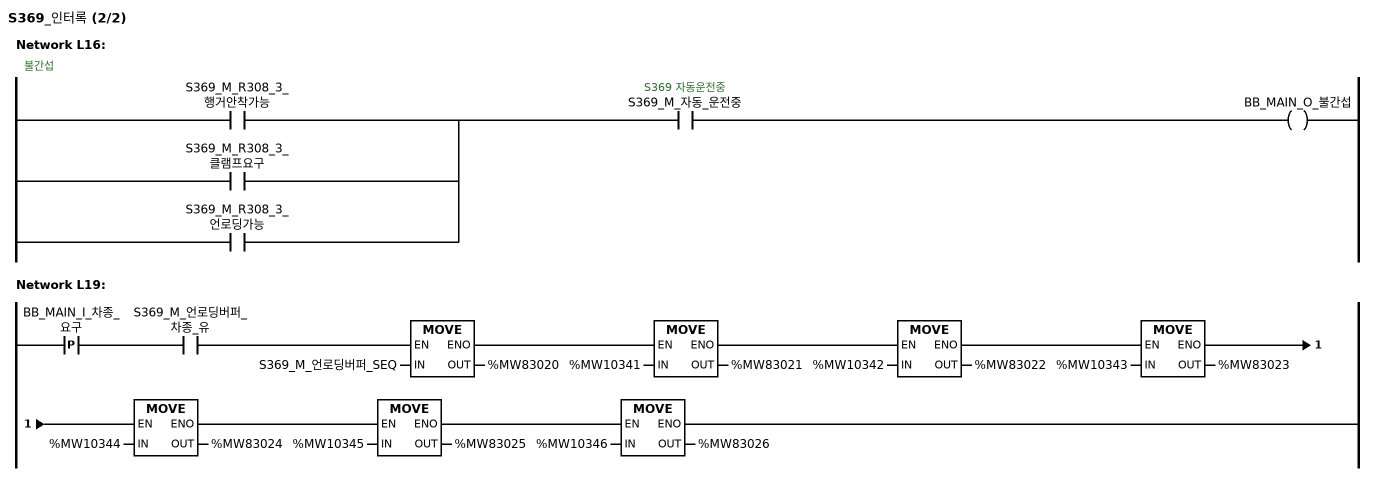
(* [picture p312: S369_인터록 rungs L16-L19] *)
(* 불간섭 *)
(* Rung L16 *)
BB_MAIN_O_불간섭 := (S369_M_R308_3_행거안착가능 OR S369_M_R308_3_클램프요구 OR S369_M_R308_3_언로딩가능) AND S369_M_자동_운전중;
(* Rung L19 *)
_e1(CLK := BB_MAIN_I_차종_요구);
IF _e1.Q AND S369_M_언로딩버퍼_차종_유 THEN
    %MW83020 := S369_M_언로딩버퍼_SEQ;
    %MW83021 := %MW10341;
    %MW83022 := %MW10342;
    %MW83023 := %MW10343;
    %MW83024 := %MW10344;
    %MW83025 := %MW10345;
    %MW83026 := %MW10346;
END_IF;
END_PROGRAM

PROGRAM S369_이상 (* task: 스캔 프로그램 *)
VAR
    INST10 : TON;
    INST11 : TON;
    INST12 : TON;
    INST13 : TON;
    INST14 : TON;
    INST15 : TON;
    INST16 : TON;
    INST17 : TON;
    INST18 : TON;
    INST19 : TON;
    INST20 : TON;
    INST21 : TON;
    INST22 : TON;
    INST23 : TON;
    INST24 : TON;
    INST25 : TON;
    INST26 : TON;
    INST27 : TON;
    INST28 : TON;
    INST29 : TON;
    INST30 : TON;
    INST31 : TON;
    INST32 : TON;
    INST33 : TON;
    INST34 : TON;
    INST35 : TON;
    INST36 : TON;
    INST37 : TON;
    INST38 : TON;
    INST8 : TON;
    INST9 : TON;
END_VAR
VAR_EXTERNAL RETAIN
    S368_M_공정_불간섭 : BOOL; (* AT %MW4004.1 *) (* S368_M_공정_불간섭 *)
    S368_M_공정_제품감지_무 : BOOL; (* AT %MW4001.6 *) (* S368_M_공정_제품감지_무 *)
    S368_M_공정_차종_유 : BOOL; (* AT %MW4002.0 *) (* S368_M_공정_차종_유 *)
    S368_M_자동_운전중 : BOOL; (* AT %MW4000.4 *) (* S368 자동운전중 *)
    S369_LOAD_M_NODE_6_41_통신_이상 : BOOL; (* AT %MW5024.0 *)
    S369_M_LD_CP_OFF : BOOL; (* AT %MW5017.0 *) (* S369_M_LD_CP_OFF *)
    S369_M_LD_EJECT_상승_LS_이상 : BOOL; (* AT %MW5100.5 *) (* S369_M_LD_EJECT_상승_LS_이상 *)
    S369_M_LD_EJECT_제품감지_이상 : BOOL; (* AT %MW5014.0 *) (* S369_M_LD_제품감지_이상 *)
    S369_M_LD_EJECT_하강_LS_이상 : BOOL; (* AT %MW5100.6 *) (* S369_M_LD_EJECT_하강_LS_이상 *)
    S369_M_LD_LH_LAT_전진_LS_이상 : BOOL; (* AT %MW5101.5 *) (* S369_M_LD_LH_LAT_전진_LS_이상 *)
    S369_M_LD_LH_LAT_후진_LS_이상 : BOOL; (* AT %MW5101.6 *) (* S369_M_LD_LH_LAT_후진_LS_이상 *)
    S369_M_LD_RH_LAT_전진_LS_이상 : BOOL; (* AT %MW5102.5 *) (* S369_M_LD_RH_LAT_전진_LS_이상 *)
    S369_M_LD_RH_LAT_후진_LS_이상 : BOOL; (* AT %MW5102.6 *) (* S369_M_LD_RH_LAT_후진_LS_이상 *)
    S369_M_LD_공기압_이상 : BOOL; (* AT %MW5013.0 *) (* S369_M_LD_공기압_이상 *)
    S369_M_LD_차종_이상 : BOOL; (* AT %MW5015.0 *) (* S369_M_LD_차종_이상 *)
    S369_M_R308_3_언로딩완료 : BOOL; (* AT %MW5001.5 *)
    S369_M_R369_2_로딩가능 : BOOL; (* AT %MW5004.8 *)
    S369_M_R369_2_로딩완료 : BOOL; (* AT %MW5001.2 *)
    S369_M_SERVO_DRIVE_통신이상 : BOOL; (* AT %MW5024.8 *)
    S369_M_SRV_NFB_OFF : BOOL; (* AT %MW5021.0 *) (* S369_M_SRV_NFB_OFF *)
    S369_M_UD_CP_OFF : BOOL; (* AT %MW5017.1 *) (* S369_M_UD_CP_OFF *)
    S369_M_UD_DOCK_CLP_전진_LS_이상 : BOOL; (* AT %MW5111.5 *) (* S369_M_UD_DOCK_CLP_전진_LS_이상 *)
    S369_M_UD_DOCK_CLP_후진_LS_이상 : BOOL; (* AT %MW5111.6 *) (* S369_M_UD_DOCK_CLP_후진_LS_이상 *)
    S369_M_UD_EJECT_상승_LS_이상 : BOOL; (* AT %MW5108.5 *) (* S369_M_UD_EJECT_상승_LS_이상 *)
    S369_M_UD_EJECT_상승단 : BOOL; (* AT %MW5108.3 *) (* S369_M_UD_EJECT_상승단 *)
    S369_M_UD_EJECT_제품감지_이상 : BOOL; (* AT %MW5014.1 *) (* S369_M_UD_제품감지_이상 *)
    S369_M_UD_EJECT_하강_LS_이상 : BOOL; (* AT %MW5108.6 *) (* S369_M_UD_EJECT_하강_LS_이상 *)
    S369_M_UD_LH_LAT_전진_LS_이상 : BOOL; (* AT %MW5109.5 *) (* S369_M_UD_LH_LAT_전진_LS_이상 *)
    S369_M_UD_LH_LAT_전진단 : BOOL; (* AT %MW5109.3 *) (* S369_M_UD_LH_LAT_전진단 *)
    S369_M_UD_LH_LAT_후진_LS_이상 : BOOL; (* AT %MW5109.6 *) (* S369_M_UD_LH_LAT_후진_LS_이상 *)
    S369_M_UD_RH_LAT_전진_LS_이상 : BOOL; (* AT %MW5110.5 *) (* S369_M_UD_RH_LAT_전진_LS_이상 *)
    S369_M_UD_RH_LAT_전진단 : BOOL; (* AT %MW5110.3 *) (* S369_M_UD_RH_LAT_전진단 *)
    S369_M_UD_RH_LAT_후진_LS_이상 : BOOL; (* AT %MW5110.6 *) (* S369_M_UD_RH_LAT_후진_LS_이상 *)
    S369_M_UD_공기압_이상 : BOOL; (* AT %MW5013.1 *) (* S369_M_UD_공기압_이상 *)
    S369_M_UD_차종_이상 : BOOL; (* AT %MW5015.1 *) (* S369_M_UD_차종_이상 *)
    S369_M_로딩_공정_불간섭 : BOOL; (* AT %MW5004.2 *) (* S369_M_공정_불간섭 *)
    S369_M_로딩_이젝터_제품감지_무 : BOOL; (* AT %MW5001.9 *)
    S369_M_로딩_이젝터_제품감지_유 : BOOL; (* AT %MW5001.8 *)
    S369_M_로딩버퍼_차종_유 : BOOL; (* AT %MW5002.0 *)
    S369_M_언로딩_공정_불간섭 : BOOL; (* AT %MW5004.3 *)
    S369_M_언로딩_이젝터_제품감지_무 : BOOL; (* AT %MW5001.11 *)
    S369_M_언로딩_이젝터_제품감지_유 : BOOL; (* AT %MW5001.10 *)
    S369_M_언로딩버퍼_차종_유 : BOOL; (* AT %MW5002.2 *)
    S369_M_이송버퍼1_제품감지_이상 : BOOL; (* AT %MW5014.5 *) (* S369_M_BELT4_제품감지_이상 *)
    S369_M_이송버퍼2_제품감지_이상 : BOOL; (* AT %MW5014.4 *) (* S369_M_BELT3_제품감지_이상 *)
    S369_M_이송버퍼3_제품감지_이상 : BOOL; (* AT %MW5014.3 *) (* S369_M_BELT2_제품감지_이상 *)
    S369_M_이송버퍼4_제품감지_이상 : BOOL; (* AT %MW5014.2 *) (* S369_M_BELT1_제품감지_이상 *)
    S369_M_자동_운전중 : BOOL; (* AT %MW5000.4 *) (* S369 자동운전중 *)
    S369_M_총괄_CP_이상 : BOOL; (* AT %MW5009.7 *) (* S369 CP OFF 이상 *)
    S369_M_총괄_CT_이상 : BOOL; (* AT %MW5010.4 *) (* S369   TACK TIME 이상 *)
    S369_M_총괄_EOCR_이상 : BOOL; (* AT %MW5009.8 *) (* S369_M_총괄_EOCR_이상 *)
    S369_M_총괄_INV_이상 : BOOL; (* AT %MW5009.9 *) (* S369_M_총괄_INV_이상 *)
    S369_M_총괄_LS_이상 : BOOL; (* AT %MW5009.15 *) (* S369 LS 이상 *)
    S369_M_총괄_MATCH_이상 : BOOL; (* AT %MW5010.0 *) (* S369 매트SW 이상 *)
    S369_M_총괄_MC_이상 : BOOL; (* AT %MW5009.13 *) (* S369_M_총괄_MC_이상 *)
    S369_M_총괄_NFB_이상 : BOOL; (* AT %MW5009.11 *) (* S369 NFB 이상 *)
    S369_M_총괄_ROBOT_이상 : BOOL; (* AT %MW5010.1 *) (* S369 ROBOT 이상 *)
    S369_M_총괄_SAFETY_이상 : BOOL; (* AT %MW5009.2 *) (* S369_M_총괄_SAFETY_이상 *)
    S369_M_총괄_SRV_이상 : BOOL; (* AT %MW5009.10 *) (* S369 SERVO 이상 *)
    S369_M_총괄_공기압_이상 : BOOL; (* AT %MW5009.3 *) (* S369 공기압 이상 *)
    S369_M_총괄_사양_이상 : BOOL; (* AT %MW5009.6 *) (* S369 사양 이상 *)
    S369_M_총괄_오버런_이상 : BOOL; (* AT %MW5009.12 *) (* S369 OVER RUN 이상 *)
    S369_M_총괄_용접타점수_이상 : BOOL; (* AT %MW5010.2 *) (* S369 용접타점수 이상 *)
    S369_M_총괄_이상 : BOOL; (* AT %MW5009.0 *) (* S369_M_총괄_이상 *)
    S369_M_총괄_제품감지_이상 : BOOL; (* AT %MW5009.4 *) (* S369 제품감지 이상 *)
    S369_M_총괄_차종_이상 : BOOL; (* AT %MW5009.5 *) (* S369 차종 이상 *)
    S369_M_총괄_통신_이상 : BOOL; (* AT %MW5009.14 *) (* S369 통신이상 *)
    S369_M_컨베어_MC_이상 : BOOL; (* AT %MW5023.0 *)
    S369_UNLD_M_NODE_6_42_통신_이상 : BOOL; (* AT %MW5024.1 *)
    전체_M_이상_리셋 : BOOL; (* AT %MW308.2 *) (* ALL공정 PB 이상리셋 *)
END_VAR
VAR_EXTERNAL
    S369LD_6_41_PLC_BOX_CP_TRIP : BOOL; (* AT %MW86412.15 *) (* S369LD_6_41_PLC_BOX_CP_TRIP *)
    S369LD_공기압_AIR_CHECK : BOOL; (* AT %MW86412.14 *) (* S369LD_공기압_AIR_CHECK *)
    S369UD_6_42_PLC_BOX_CP_TRIP : BOOL; (* AT %MW86422.15 *) (* S369UD_6_42_PLC_BOX_CP_TRIP *)
    S369UD_공기압_AIR_CHECK : BOOL; (* AT %MW86422.14 *) (* S369UD_공기압_AIR_CHECK *)
    S369_CONVEY_I_서보드라이브_이상 : BOOL; (* AT %MW50000.8 *)
    S369_SERVO_MC_ON : BOOL; (* AT %MW85022.0 *) (* SERVO_BRAKE_ON *)
    S369_SERVO_NFB_ON : BOOL; (* AT %MW85023.0 *)
    SERVO_SAFETY_CR_ON : BOOL; (* AT %MW95024.0 *) (* SERVO_BRAKE_CR_ON *)
    _0005_EB63_S00_SVC_ER : BOOL; (* AT %MW185036.7 *) (* 통신 서비스 에러 *)
    _0006_EB41_CFG_ER : BOOL; (* AT %MW186064.0 *) (* EB 구성 에러 *)
    _0006_EB41_DEER : BOOL; (* AT %MW186064.1 *) (* EB 운전 중 탈락 *)
    _0006_EB41_IO_DEER : BOOL; (* AT %MW186065.2 *) (* EB IO 탈락 에러 *)
    _0006_EB41_IO_TYER : BOOL; (* AT %MW186065.1 *) (* EB IO 타입 에러 *)
    _0006_EB42_CFG_ER : BOOL; (* AT %MW186070.0 *) (* EB 구성 에러 *)
    _0006_EB42_DEER : BOOL; (* AT %MW186070.1 *) (* EB 운전 중 탈락 *)
    _0006_EB42_IO_DEER : BOOL; (* AT %MW186071.2 *) (* EB IO 탈락 에러 *)
    _0006_EB42_IO_TYER : BOOL; (* AT %MW186071.1 *) (* EB IO 타입 에러 *)
    _0007_EB10_CFG_ER : BOOL; (* AT %MW187040.0 *) (* EB 구성 에러 *)
    _0007_EB10_DEER : BOOL; (* AT %MW187040.1 *) (* EB 운전 중 탈락 *)
    _0007_EB10_IO_DEER : BOOL; (* AT %MW187041.2 *) (* EB IO 탈락 에러 *)
    _0007_EB10_IO_TYER : BOOL; (* AT %MW187041.1 *) (* EB IO 타입 에러 *)
END_VAR

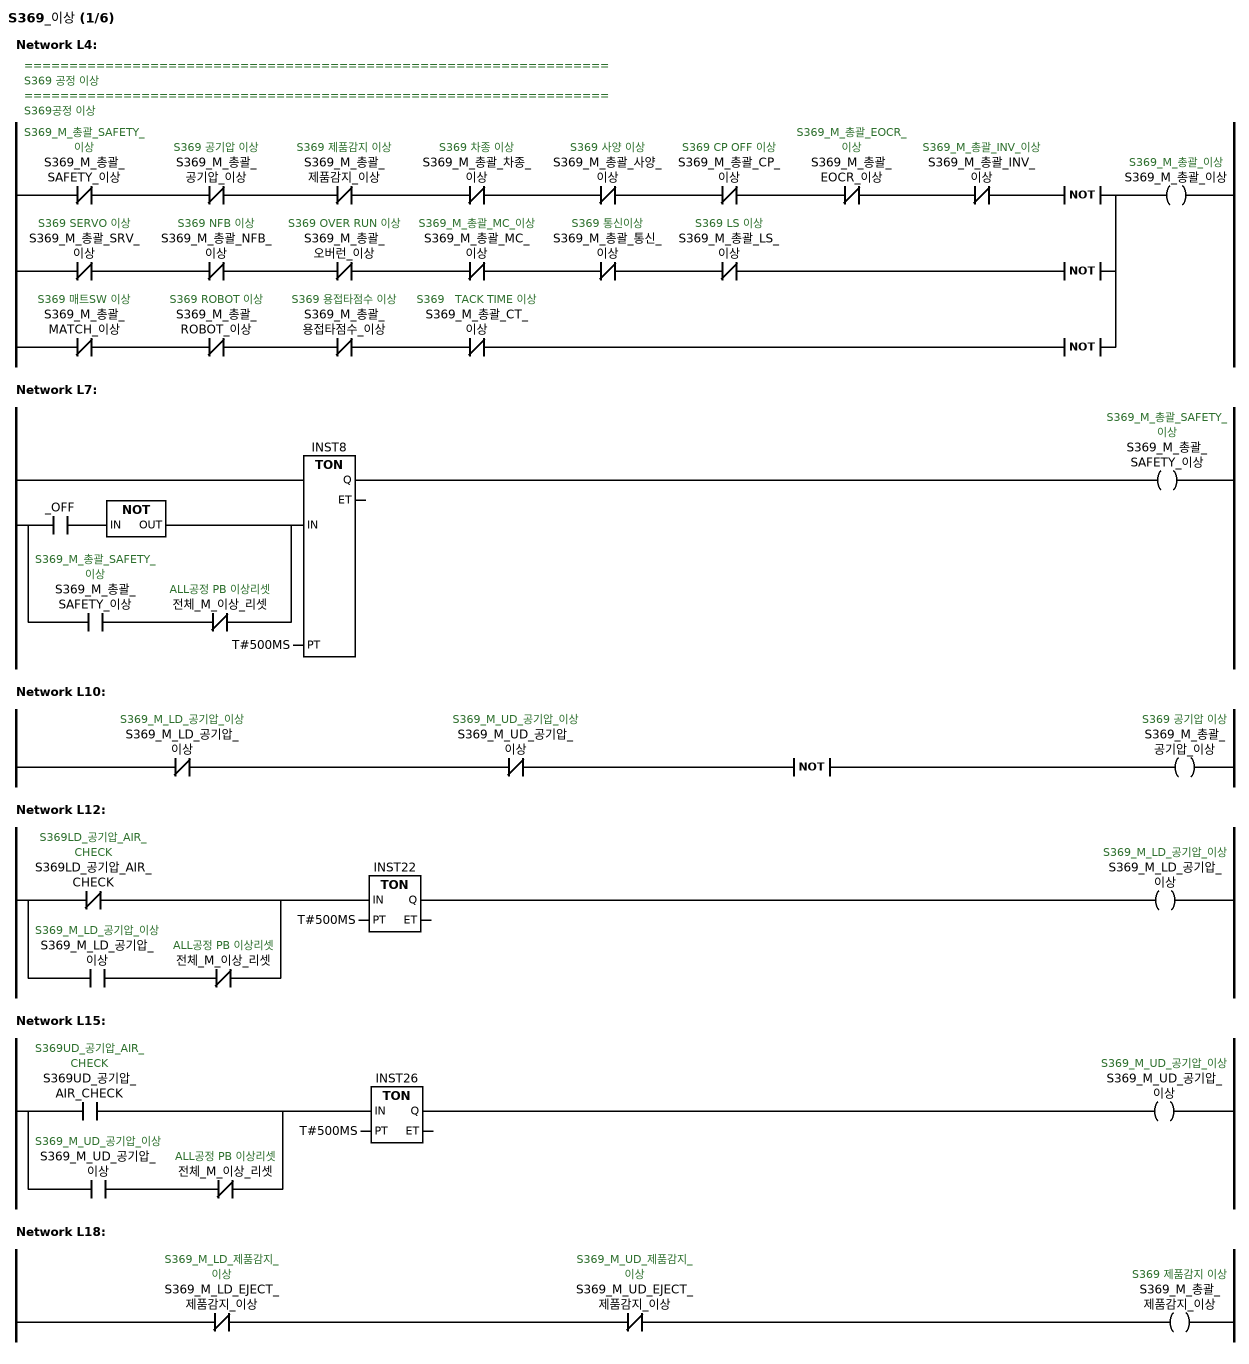
(* ================================================================= *)
(* S369 공정 이상 *)
(* ================================================================= *)
(* S369공정 이상 *)
(* Rung L4 *)
S369_M_총괄_이상 := NOT (NOT S369_M_총괄_SAFETY_이상 AND NOT S369_M_총괄_공기압_이상 AND NOT S369_M_총괄_제품감지_이상 AND NOT S369_M_총괄_차종_이상 AND NOT S369_M_총괄_사양_이상 AND NOT S369_M_총괄_CP_이상 AND NOT S369_M_총괄_EOCR_이상 AND NOT S369_M_총괄_INV_이상) OR NOT (NOT S369_M_총괄_SRV_이상 AND NOT S369_M_총괄_NFB_이상 AND NOT S369_M_총괄_오버런_이상 AND NOT S369_M_총괄_MC_이상 AND NOT S369_M_총괄_통신_이상 AND NOT S369_M_총괄_LS_이상) OR NOT (NOT S369_M_총괄_MATCH_이상 AND NOT S369_M_총괄_ROBOT_이상 AND NOT S369_M_총괄_용접타점수_이상 AND NOT S369_M_총괄_CT_이상);
(* Rung L7 *)
INST8(IN := (NOT _OFF) OR (S369_M_총괄_SAFETY_이상 AND NOT 전체_M_이상_리셋), PT := T#500MS);
S369_M_총괄_SAFETY_이상 := INST8.Q;
(* Rung L10 *)
S369_M_총괄_공기압_이상 := NOT (NOT S369_M_LD_공기압_이상 AND NOT S369_M_UD_공기압_이상);
(* Rung L12 *)
INST22(IN := NOT S369LD_공기압_AIR_CHECK OR (S369_M_LD_공기압_이상 AND NOT 전체_M_이상_리셋), PT := T#500MS);
S369_M_LD_공기압_이상 := INST22.Q;
(* Rung L15 *)
INST26(IN := S369UD_공기압_AIR_CHECK OR (S369_M_UD_공기압_이상 AND NOT 전체_M_이상_리셋), PT := T#500MS);
S369_M_UD_공기압_이상 := INST26.Q;
(* Rung L18 *)
S369_M_총괄_제품감지_이상 := NOT S369_M_LD_EJECT_제품감지_이상 AND NOT S369_M_UD_EJECT_제품감지_이상;

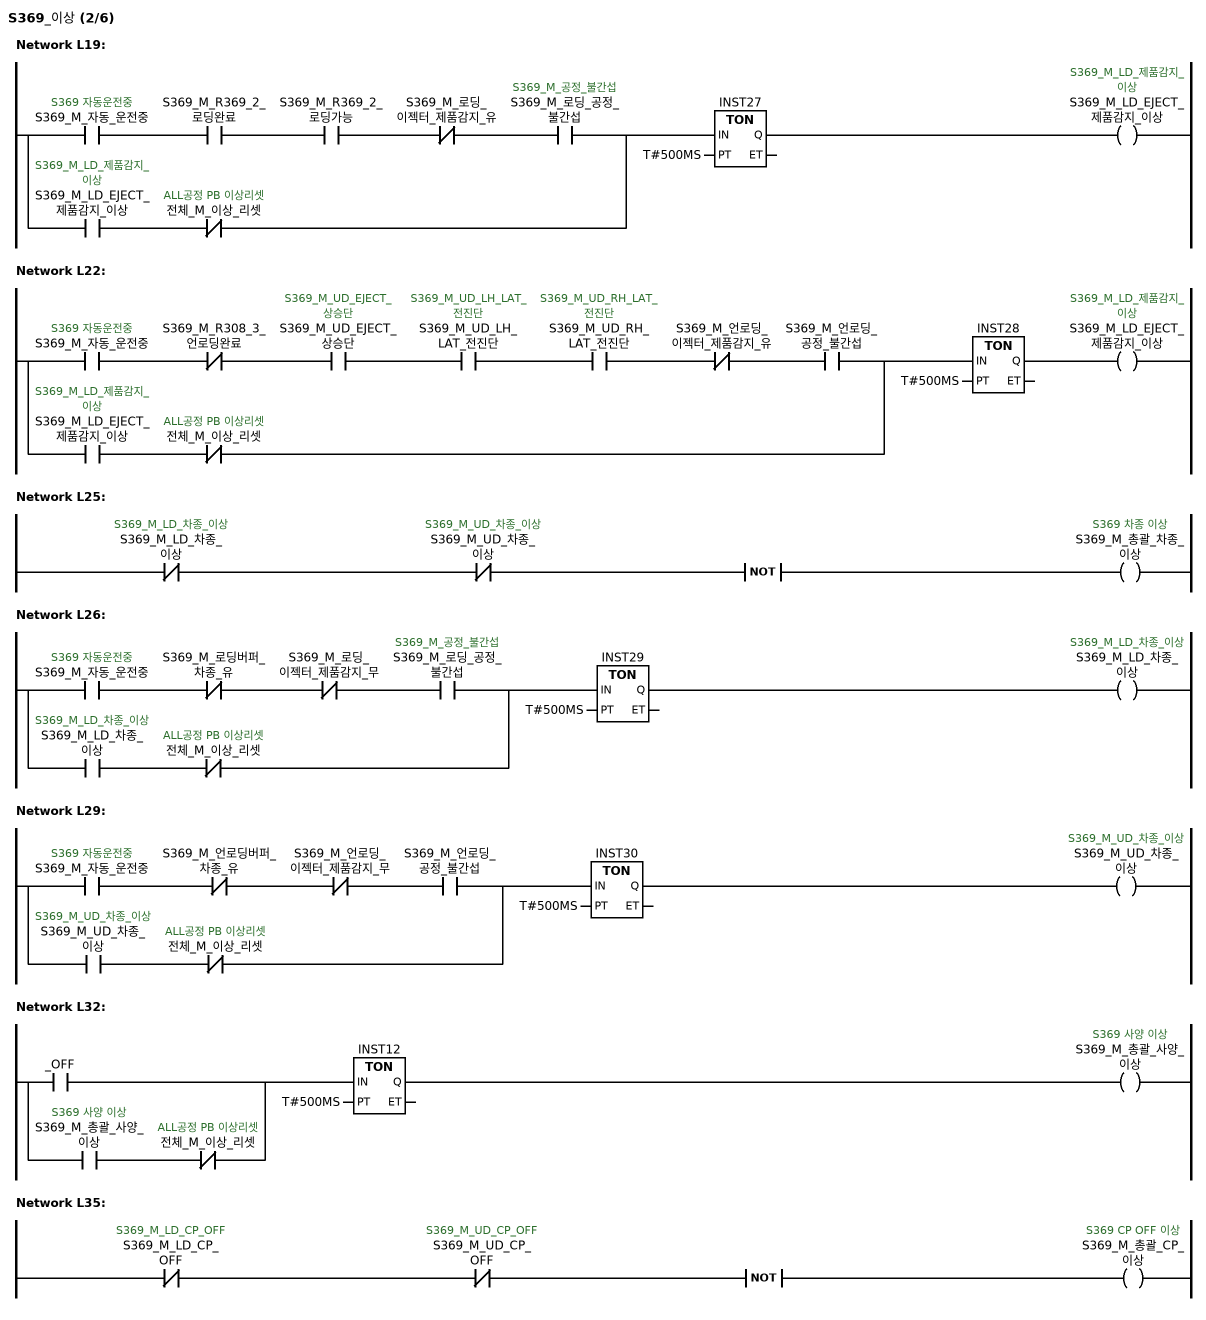
(* Rung L19 *)
INST27(IN := (S369_M_자동_운전중 AND S369_M_R369_2_로딩완료 AND S369_M_R369_2_로딩가능 AND NOT S369_M_로딩_이젝터_제품감지_유 AND S369_M_로딩_공정_불간섭) OR (S369_M_LD_EJECT_제품감지_이상 AND NOT 전체_M_이상_리셋), PT := T#500MS);
S369_M_LD_EJECT_제품감지_이상 := INST27.Q;
(* Rung L22 *)
INST28(IN := (S369_M_자동_운전중 AND NOT S369_M_R308_3_언로딩완료 AND S369_M_UD_EJECT_상승단 AND S369_M_UD_LH_LAT_전진단 AND S369_M_UD_RH_LAT_전진단 AND NOT S369_M_언로딩_이젝터_제품감지_유 AND S369_M_언로딩_공정_불간섭) OR (S369_M_LD_EJECT_제품감지_이상 AND NOT 전체_M_이상_리셋), PT := T#500MS);
S369_M_LD_EJECT_제품감지_이상 := INST28.Q;
(* Rung L25 *)
S369_M_총괄_차종_이상 := NOT (NOT S369_M_LD_차종_이상 AND NOT S369_M_UD_차종_이상);
(* Rung L26 *)
INST29(IN := (S369_M_자동_운전중 AND NOT S369_M_로딩버퍼_차종_유 AND NOT S369_M_로딩_이젝터_제품감지_무 AND S369_M_로딩_공정_불간섭) OR (S369_M_LD_차종_이상 AND NOT 전체_M_이상_리셋), PT := T#500MS);
S369_M_LD_차종_이상 := INST29.Q;
(* Rung L29 *)
INST30(IN := (S369_M_자동_운전중 AND NOT S369_M_언로딩버퍼_차종_유 AND NOT S369_M_언로딩_이젝터_제품감지_무 AND S369_M_언로딩_공정_불간섭) OR (S369_M_UD_차종_이상 AND NOT 전체_M_이상_리셋), PT := T#500MS);
S369_M_UD_차종_이상 := INST30.Q;
(* Rung L32 *)
INST12(IN := _OFF OR (S369_M_총괄_사양_이상 AND NOT 전체_M_이상_리셋), PT := T#500MS);
S369_M_총괄_사양_이상 := INST12.Q;
(* Rung L35 *)
S369_M_총괄_CP_이상 := NOT (NOT S369_M_LD_CP_OFF AND NOT S369_M_UD_CP_OFF);

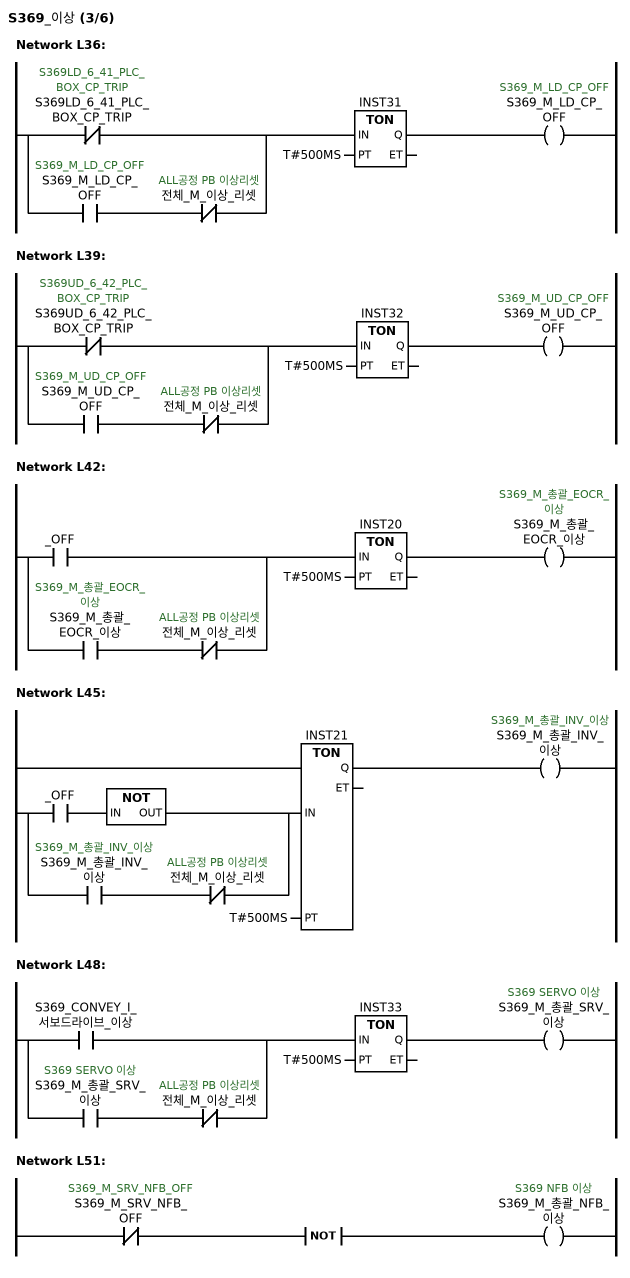
(* Rung L36 *)
INST31(IN := NOT S369LD_6_41_PLC_BOX_CP_TRIP OR (S369_M_LD_CP_OFF AND NOT 전체_M_이상_리셋), PT := T#500MS);
S369_M_LD_CP_OFF := INST31.Q;
(* Rung L39 *)
INST32(IN := NOT S369UD_6_42_PLC_BOX_CP_TRIP OR (S369_M_UD_CP_OFF AND NOT 전체_M_이상_리셋), PT := T#500MS);
S369_M_UD_CP_OFF := INST32.Q;
(* Rung L42 *)
INST20(IN := _OFF OR (S369_M_총괄_EOCR_이상 AND NOT 전체_M_이상_리셋), PT := T#500MS);
S369_M_총괄_EOCR_이상 := INST20.Q;
(* Rung L45 *)
INST21(IN := (NOT _OFF) OR (S369_M_총괄_INV_이상 AND NOT 전체_M_이상_리셋), PT := T#500MS);
S369_M_총괄_INV_이상 := INST21.Q;
(* Rung L48 *)
INST33(IN := S369_CONVEY_I_서보드라이브_이상 OR (S369_M_총괄_SRV_이상 AND NOT 전체_M_이상_리셋), PT := T#500MS);
S369_M_총괄_SRV_이상 := INST33.Q;
(* Rung L51 *)
S369_M_총괄_NFB_이상 := S369_M_SRV_NFB_OFF;

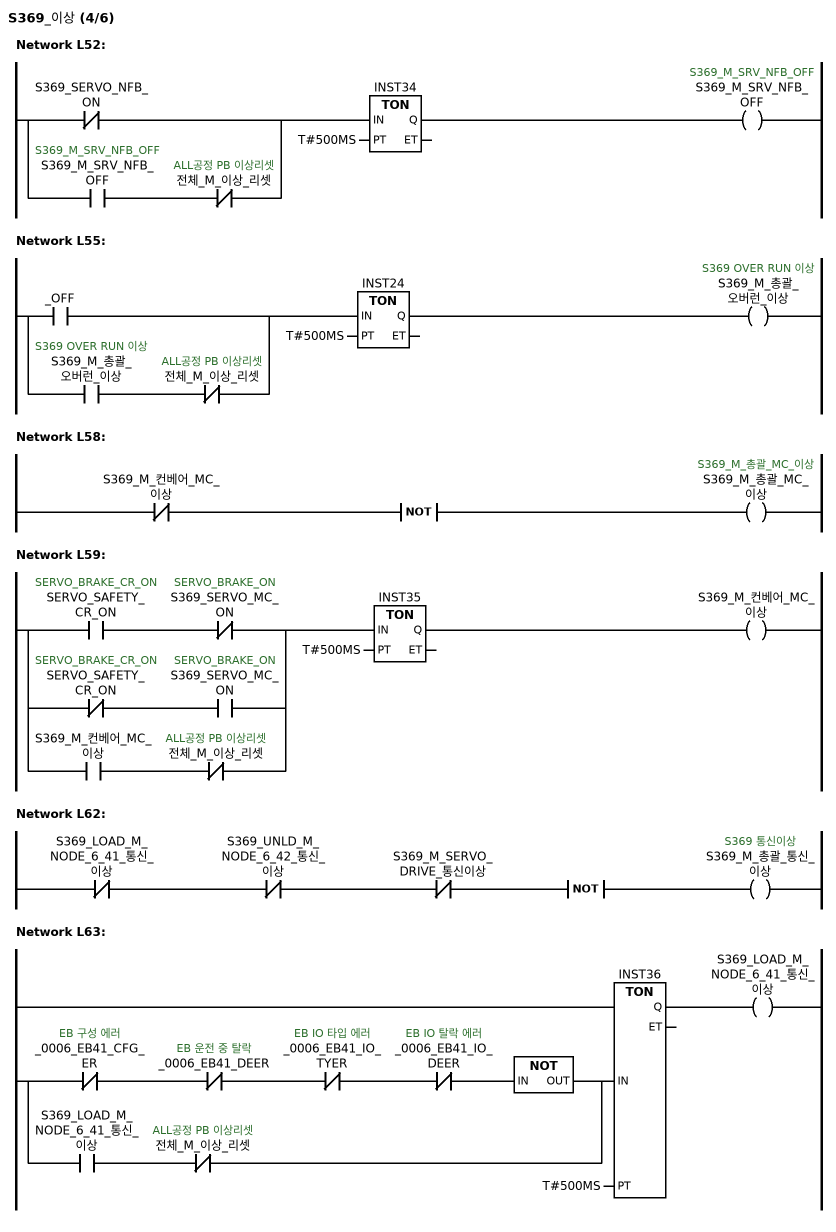
(* Rung L52 *)
INST34(IN := NOT S369_SERVO_NFB_ON OR (S369_M_SRV_NFB_OFF AND NOT 전체_M_이상_리셋), PT := T#500MS);
S369_M_SRV_NFB_OFF := INST34.Q;
(* Rung L55 *)
INST24(IN := _OFF OR (S369_M_총괄_오버런_이상 AND NOT 전체_M_이상_리셋), PT := T#500MS);
S369_M_총괄_오버런_이상 := INST24.Q;
(* Rung L58 *)
S369_M_총괄_MC_이상 := S369_M_컨베어_MC_이상;
(* Rung L59 *)
INST35(IN := (SERVO_SAFETY_CR_ON AND NOT S369_SERVO_MC_ON) OR (NOT SERVO_SAFETY_CR_ON AND S369_SERVO_MC_ON) OR (S369_M_컨베어_MC_이상 AND NOT 전체_M_이상_리셋), PT := T#500MS);
S369_M_컨베어_MC_이상 := INST35.Q;
(* Rung L62 *)
S369_M_총괄_통신_이상 := NOT (NOT S369_LOAD_M_NODE_6_41_통신_이상 AND NOT S369_UNLD_M_NODE_6_42_통신_이상 AND NOT S369_M_SERVO_DRIVE_통신이상);
(* Rung L63 *)
INST36(IN := (NOT (NOT _0006_EB41_CFG_ER AND NOT _0006_EB41_DEER AND NOT _0006_EB41_IO_TYER AND NOT _0006_EB41_IO_DEER)) OR (S369_LOAD_M_NODE_6_41_통신_이상 AND NOT 전체_M_이상_리셋), PT := T#500MS);
S369_LOAD_M_NODE_6_41_통신_이상 := INST36.Q;

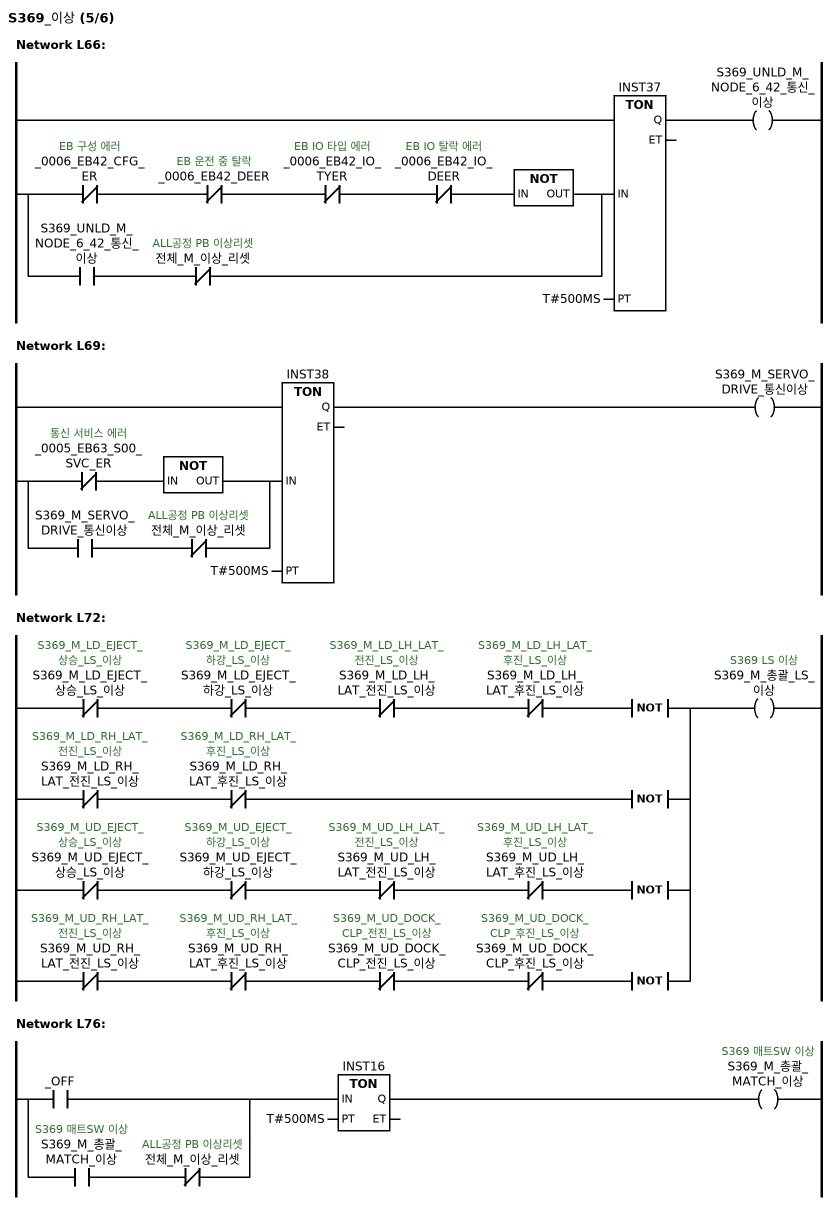
(* Rung L66 *)
INST37(IN := (NOT (NOT _0006_EB42_CFG_ER AND NOT _0006_EB42_DEER AND NOT _0006_EB42_IO_TYER AND NOT _0006_EB42_IO_DEER)) OR (S369_UNLD_M_NODE_6_42_통신_이상 AND NOT 전체_M_이상_리셋), PT := T#500MS);
S369_UNLD_M_NODE_6_42_통신_이상 := INST37.Q;
(* Rung L69 *)
INST38(IN := (NOT (NOT _0005_EB63_S00_SVC_ER)) OR (S369_M_SERVO_DRIVE_통신이상 AND NOT 전체_M_이상_리셋), PT := T#500MS);
S369_M_SERVO_DRIVE_통신이상 := INST38.Q;
(* Rung L72 *)
S369_M_총괄_LS_이상 := NOT (NOT S369_M_LD_EJECT_상승_LS_이상 AND NOT S369_M_LD_EJECT_하강_LS_이상 AND NOT S369_M_LD_LH_LAT_전진_LS_이상 AND NOT S369_M_LD_LH_LAT_후진_LS_이상) OR NOT (NOT S369_M_LD_RH_LAT_전진_LS_이상 AND NOT S369_M_LD_RH_LAT_후진_LS_이상) OR NOT (NOT S369_M_UD_EJECT_상승_LS_이상 AND NOT S369_M_UD_EJECT_하강_LS_이상 AND NOT S369_M_UD_LH_LAT_전진_LS_이상 AND NOT S369_M_UD_LH_LAT_후진_LS_이상) OR NOT (NOT S369_M_UD_RH_LAT_전진_LS_이상 AND NOT S369_M_UD_RH_LAT_후진_LS_이상 AND NOT S369_M_UD_DOCK_CLP_전진_LS_이상 AND NOT S369_M_UD_DOCK_CLP_후진_LS_이상);
(* Rung L76 *)
INST16(IN := _OFF OR (S369_M_총괄_MATCH_이상 AND NOT 전체_M_이상_리셋), PT := T#500MS);
S369_M_총괄_MATCH_이상 := INST16.Q;

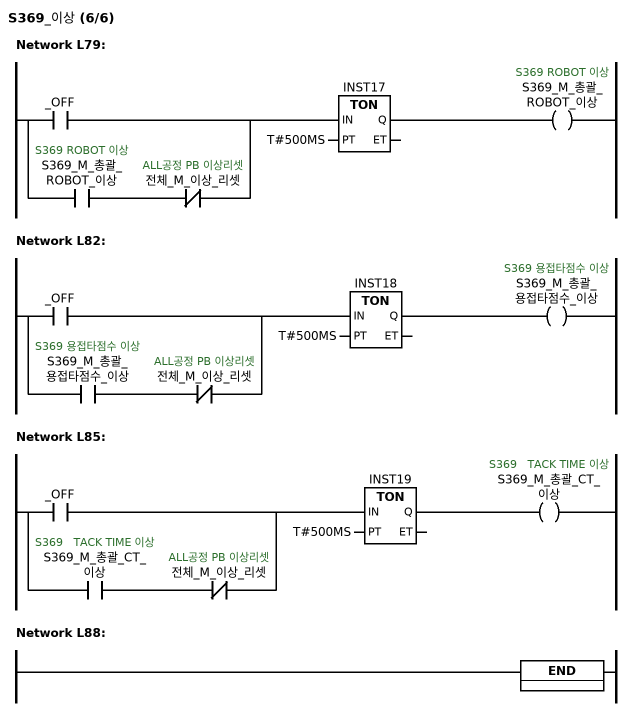
(* Rung L79 *)
INST17(IN := _OFF OR (S369_M_총괄_ROBOT_이상 AND NOT 전체_M_이상_리셋), PT := T#500MS);
S369_M_총괄_ROBOT_이상 := INST17.Q;
(* Rung L82 *)
INST18(IN := _OFF OR (S369_M_총괄_용접타점수_이상 AND NOT 전체_M_이상_리셋), PT := T#500MS);
S369_M_총괄_용접타점수_이상 := INST18.Q;
(* Rung L85 *)
INST19(IN := _OFF OR (S369_M_총괄_CT_이상 AND NOT 전체_M_이상_리셋), PT := T#500MS);
S369_M_총괄_CT_이상 := INST19.Q;
(* Rung L88 *)
END();
END_PROGRAM

PROGRAM HMI_차종수정 (* task: 스캔 프로그램 *)
VAR_EXTERNAL RETAIN
    CARTYPE : ARRAY[0..599] OF WORD; (* AT %MW10000 *) (* CARTYPE *)
    HMI_M_매칭_R361_1_S366 : BOOL; (* AT %MW70.0 *)
    HMI_M_매칭_S366_R361_1 : BOOL; (* AT %MW70.1 *)
    HMI_M_매칭선택 : WORD; (* AT %MW70 *)
    HMI_M_매칭차종_DATA_OK : BOOL; (* AT %MW9.9 *)
    HMI_M_매칭차종_복사_ON : BOOL; (* AT %MW9.6 *)
    HMI_M_매칭차종_복사_SET : BOOL; (* AT %MW9.8 *)
    HMI_M_차종매칭_SEQ : WORD; (* AT %MW50 *)
    HMI_M_차종매칭_차종1_AX : BOOL; (* AT %MW51.0 *)
    HMI_M_차종매칭_차종1_B : BOOL; (* AT %MW51.1 *)
    HMI_M_차종매칭_차종1_C : BOOL; (* AT %MW51.2 *)
    HMI_M_차종매칭_차종1_D : BOOL; (* AT %MW51.3 *)
    HMI_M_차종매칭_차종1_E : BOOL; (* AT %MW51.4 *)
    HMI_M_차종매칭_차종1_F : BOOL; (* AT %MW51.5 *)
    HMI_M_차종매칭_차종1_G : BOOL; (* AT %MW51.6 *)
    HMI_M_차종매칭_차종1_H : BOOL; (* AT %MW51.7 *)
    HMI_M_차종매칭_차종2_3DR : BOOL; (* AT %MW51.8 *)
    HMI_M_차종매칭_차종2_4DR : BOOL; (* AT %MW51.9 *)
    HMI_M_차종매칭_차종2_5DR : BOOL; (* AT %MW51.10 *)
    HMI_M_차종매칭_차종2_SP1 : BOOL; (* AT %MW51.12 *)
    HMI_M_차종매칭_차종2_SP2 : BOOL; (* AT %MW51.13 *)
    HMI_M_차종매칭_차종2_WGN : BOOL; (* AT %MW51.11 *)
    HMI_M_차종매칭_차종3_LHD : BOOL; (* AT %MW51.14 *)
    HMI_M_차종매칭_차종3_RHD : BOOL; (* AT %MW51.15 *)
    HMI_M_차종매칭_차종4_EEC : BOOL; (* AT %MW52.3 *)
    HMI_M_차종매칭_차종4_SP1 : BOOL; (* AT %MW52.8 *)
    HMI_M_차종매칭_차종4_SP2 : BOOL; (* AT %MW52.9 *)
    HMI_M_차종매칭_차종4_SP3 : BOOL; (* AT %MW52.11 *)
    HMI_M_차종매칭_차종4_SP4 : BOOL; (* AT %MW52.12 *)
    HMI_M_차종매칭_차종4_SP5 : BOOL; (* AT %MW52.13 *)
    HMI_M_차종매칭_차종4_SP6 : BOOL; (* AT %MW52.14 *)
    HMI_M_차종매칭_차종4_SP7 : BOOL; (* AT %MW52.15 *)
    HMI_M_차종매칭_차종4_내수 : BOOL; (* AT %MW52.0 *)
    HMI_M_차종매칭_차종4_러시아 : BOOL; (* AT %MW52.10 *)
    HMI_M_차종매칭_차종4_북미 : BOOL; (* AT %MW52.2 *)
    HMI_M_차종매칭_차종4_브라질 : BOOL; (* AT %MW52.7 *)
    HMI_M_차종매칭_차종4_수출 : BOOL; (* AT %MW52.1 *)
    HMI_M_차종매칭_차종4_중국 : BOOL; (* AT %MW52.6 *)
    HMI_M_차종매칭_차종4_중동 : BOOL; (* AT %MW52.5 *)
    HMI_M_차종매칭_차종4_호주 : BOOL; (* AT %MW52.4 *)
    HMI_M_차종매칭_차종5_AT : BOOL; (* AT %MW53.1 *)
    HMI_M_차종매칭_차종5_MT : BOOL; (* AT %MW53.0 *)
    HMI_M_차종매칭_차종5_SP1 : BOOL; (* AT %MW53.2 *)
    HMI_M_차종매칭_차종6_DSROOF : BOOL; (* AT %MW53.6 *)
    HMI_M_차종매칭_차종6_SP1 : BOOL; (* AT %MW53.7 *)
    HMI_M_차종매칭_차종6_썬루프 : BOOL; (* AT %MW53.4 *)
    HMI_M_차종매칭_차종6_일반루프 : BOOL; (* AT %MW53.3 *)
    HMI_M_차종매칭_차종6_파노라마루프 : BOOL; (* AT %MW53.5 *)
    HMI_M_차종매칭_차종7_DSL : BOOL; (* AT %MW53.9 *)
    HMI_M_차종매칭_차종7_GSL : BOOL; (* AT %MW53.8 *)
    HMI_M_차종매칭_차종7_SP1 : BOOL; (* AT %MW53.10 *)
    HMI_M_차종매칭_차종7_SP2 : BOOL; (* AT %MW53.11 *)
    HMI_M_차종매칭_차종7_SP3 : BOOL; (* AT %MW53.12 *)
    HMI_M_차종매칭_차종7_SP4 : BOOL; (* AT %MW53.13 *)
    HMI_M_차종매칭_차종7_SP5 : BOOL; (* AT %MW53.14 *)
    HMI_M_차종매칭_차종7_SP6 : BOOL; (* AT %MW53.15 *)
    HMI_M_차종매칭_차종8_2WD : BOOL; (* AT %MW54.0 *)
    HMI_M_차종매칭_차종8_4WD : BOOL; (* AT %MW54.1 *)
    HMI_M_차종매칭_차종8_SP1 : BOOL; (* AT %MW54.2 *)
    HMI_M_차종매칭_차종9_MPI : BOOL; (* AT %MW54.3 *)
    HMI_M_차종매칭_차종9_SP1 : BOOL; (* AT %MW54.5 *)
    HMI_M_차종매칭_차종9_SP10 : BOOL; (* AT %MW54.14 *)
    HMI_M_차종매칭_차종9_SP11 : BOOL; (* AT %MW54.15 *)
    HMI_M_차종매칭_차종9_SP2 : BOOL; (* AT %MW54.6 *)
    HMI_M_차종매칭_차종9_SP3 : BOOL; (* AT %MW54.7 *)
    HMI_M_차종매칭_차종9_SP4 : BOOL; (* AT %MW54.8 *)
    HMI_M_차종매칭_차종9_SP5 : BOOL; (* AT %MW54.9 *)
    HMI_M_차종매칭_차종9_SP6 : BOOL; (* AT %MW54.10 *)
    HMI_M_차종매칭_차종9_SP7 : BOOL; (* AT %MW54.11 *)
    HMI_M_차종매칭_차종9_SP8 : BOOL; (* AT %MW54.12 *)
    HMI_M_차종매칭_차종9_SP9 : BOOL; (* AT %MW54.13 *)
    HMI_M_차종매칭_차종9_T_GDI : BOOL; (* AT %MW54.4 *)
    HMI_M_차종매칭_차종_OPT1_R_RACK_무 : BOOL; (* AT %MW55.3 *)
    HMI_M_차종매칭_차종_OPT1_R_RACK_유 : BOOL; (* AT %MW55.2 *)
    HMI_M_차종매칭_차종_OPT1_S_REP_EATER_무 : BOOL; (* AT %MW55.7 *)
    HMI_M_차종매칭_차종_OPT1_S_REP_EATER_유 : BOOL; (* AT %MW55.6 *)
    HMI_M_차종매칭_차종_OPT1_VAN_무 : BOOL; (* AT %MW55.9 *)
    HMI_M_차종매칭_차종_OPT1_VAN_유 : BOOL; (* AT %MW55.8 *)
    HMI_M_차종매칭_차종_OPT1_슬라이딩_무 : BOOL; (* AT %MW55.1 *)
    HMI_M_차종매칭_차종_OPT1_슬라이딩_유 : BOOL; (* AT %MW55.0 *)
    HMI_M_차종매칭_차종_OPT1_폴딩_무 : BOOL; (* AT %MW55.5 *)
    HMI_M_차종매칭_차종_OPT1_폴딩_유 : BOOL; (* AT %MW55.4 *)
    HMI_M_차종매칭_차종_공대차 : BOOL; (* AT %MW60.12 *)
    HMI_M_차종매칭_차종_공차 : BOOL; (* AT %MW60.10 *)
    HMI_M_차종매칭_차종_불량대차 : BOOL; (* AT %MW60.13 *)
    HMI_M_차종매칭_차종_불량차 : BOOL; (* AT %MW60.11 *)
    HMI_M_차종수정 : ARRAY[0..19] OF WORD; (* AT %MW10 *)
    HMI_M_차종수정_DATA_OK : BOOL; (* AT %MW9.0 *)
    HMI_M_차종수정_RESET : BOOL; (* AT %MW9.2 *)
    HMI_M_차종수정_SEQ : WORD; (* AT %MW10 *)
    HMI_M_차종수정_SET : BOOL; (* AT %MW9.1 *)
    HMI_M_차종수정_차종1_AX : BOOL; (* AT %MW11.0 *)
    HMI_M_차종수정_차종1_B : BOOL; (* AT %MW11.1 *)
    HMI_M_차종수정_차종1_C : BOOL; (* AT %MW11.2 *)
    HMI_M_차종수정_차종1_D : BOOL; (* AT %MW11.3 *)
    HMI_M_차종수정_차종1_E : BOOL; (* AT %MW11.4 *)
    HMI_M_차종수정_차종1_F : BOOL; (* AT %MW11.5 *)
    HMI_M_차종수정_차종1_G : BOOL; (* AT %MW11.6 *)
    HMI_M_차종수정_차종1_H : BOOL; (* AT %MW11.7 *)
    HMI_M_차종수정_차종2_3DR : BOOL; (* AT %MW11.8 *)
    HMI_M_차종수정_차종2_4DR : BOOL; (* AT %MW11.9 *)
    HMI_M_차종수정_차종2_5DR : BOOL; (* AT %MW11.10 *)
    HMI_M_차종수정_차종2_SP1 : BOOL; (* AT %MW11.12 *)
    HMI_M_차종수정_차종2_SP2 : BOOL; (* AT %MW11.13 *)
    HMI_M_차종수정_차종2_WGN : BOOL; (* AT %MW11.11 *)
    HMI_M_차종수정_차종3_LHD : BOOL; (* AT %MW11.14 *)
    HMI_M_차종수정_차종3_RHD : BOOL; (* AT %MW11.15 *)
    HMI_M_차종수정_차종4_EEC : BOOL; (* AT %MW12.3 *)
    HMI_M_차종수정_차종4_SP1 : BOOL; (* AT %MW12.8 *)
    HMI_M_차종수정_차종4_SP2 : BOOL; (* AT %MW12.9 *)
    HMI_M_차종수정_차종4_SP3 : BOOL; (* AT %MW12.11 *)
    HMI_M_차종수정_차종4_SP4 : BOOL; (* AT %MW12.12 *)
    HMI_M_차종수정_차종4_SP5 : BOOL; (* AT %MW12.13 *)
    HMI_M_차종수정_차종4_SP6 : BOOL; (* AT %MW12.14 *)
    HMI_M_차종수정_차종4_SP7 : BOOL; (* AT %MW12.15 *)
    HMI_M_차종수정_차종4_내수 : BOOL; (* AT %MW12.0 *)
    HMI_M_차종수정_차종4_러시아 : BOOL; (* AT %MW12.10 *)
    HMI_M_차종수정_차종4_북미 : BOOL; (* AT %MW12.2 *)
    HMI_M_차종수정_차종4_브라질 : BOOL; (* AT %MW12.7 *)
    HMI_M_차종수정_차종4_수출 : BOOL; (* AT %MW12.1 *)
    HMI_M_차종수정_차종4_중국 : BOOL; (* AT %MW12.6 *)
    HMI_M_차종수정_차종4_중동 : BOOL; (* AT %MW12.5 *)
    HMI_M_차종수정_차종4_호주 : BOOL; (* AT %MW12.4 *)
    HMI_M_차종수정_차종5_AT : BOOL; (* AT %MW13.1 *)
    HMI_M_차종수정_차종5_MT : BOOL; (* AT %MW13.0 *)
    HMI_M_차종수정_차종5_SP1 : BOOL; (* AT %MW13.2 *)
    HMI_M_차종수정_차종6_DSROOF : BOOL; (* AT %MW13.6 *)
    HMI_M_차종수정_차종6_SP1 : BOOL; (* AT %MW13.7 *)
    HMI_M_차종수정_차종6_썬루프 : BOOL; (* AT %MW13.4 *)
    HMI_M_차종수정_차종6_일반루프 : BOOL; (* AT %MW13.3 *)
    HMI_M_차종수정_차종6_파노라마루프 : BOOL; (* AT %MW13.5 *)
    HMI_M_차종수정_차종7_DSL : BOOL; (* AT %MW13.9 *)
    HMI_M_차종수정_차종7_GSL : BOOL; (* AT %MW13.8 *)
    HMI_M_차종수정_차종7_SP1 : BOOL; (* AT %MW13.10 *)
    HMI_M_차종수정_차종7_SP2 : BOOL; (* AT %MW13.11 *)
    HMI_M_차종수정_차종7_SP3 : BOOL; (* AT %MW13.12 *)
    HMI_M_차종수정_차종7_SP4 : BOOL; (* AT %MW13.13 *)
    HMI_M_차종수정_차종7_SP5 : BOOL; (* AT %MW13.14 *)
    HMI_M_차종수정_차종7_SP6 : BOOL; (* AT %MW13.15 *)
    HMI_M_차종수정_차종8_2WD : BOOL; (* AT %MW14.0 *)
    HMI_M_차종수정_차종8_4WD : BOOL; (* AT %MW14.1 *)
    HMI_M_차종수정_차종8_SP1 : BOOL; (* AT %MW14.2 *)
    HMI_M_차종수정_차종9_MPI : BOOL; (* AT %MW14.3 *)
    HMI_M_차종수정_차종9_SP1 : BOOL; (* AT %MW14.5 *)
    HMI_M_차종수정_차종9_SP10 : BOOL; (* AT %MW14.14 *)
    HMI_M_차종수정_차종9_SP11 : BOOL; (* AT %MW14.15 *)
    HMI_M_차종수정_차종9_SP2 : BOOL; (* AT %MW14.6 *)
    HMI_M_차종수정_차종9_SP3 : BOOL; (* AT %MW14.7 *)
    HMI_M_차종수정_차종9_SP4 : BOOL; (* AT %MW14.8 *)
    HMI_M_차종수정_차종9_SP5 : BOOL; (* AT %MW14.9 *)
    HMI_M_차종수정_차종9_SP6 : BOOL; (* AT %MW14.10 *)
    HMI_M_차종수정_차종9_SP7 : BOOL; (* AT %MW14.11 *)
    HMI_M_차종수정_차종9_SP8 : BOOL; (* AT %MW14.12 *)
    HMI_M_차종수정_차종9_SP9 : BOOL; (* AT %MW14.13 *)
    HMI_M_차종수정_차종9_T_GDI : BOOL; (* AT %MW14.4 *)
    HMI_M_차종수정_차종_OPT1_R_RACK_무 : BOOL; (* AT %MW15.3 *)
    HMI_M_차종수정_차종_OPT1_R_RACK_유 : BOOL; (* AT %MW15.2 *)
    HMI_M_차종수정_차종_OPT1_S_REP_EATER_무 : BOOL; (* AT %MW15.7 *)
    HMI_M_차종수정_차종_OPT1_S_REP_EATER_유 : BOOL; (* AT %MW15.6 *)
    HMI_M_차종수정_차종_OPT1_VAN_무 : BOOL; (* AT %MW15.9 *)
    HMI_M_차종수정_차종_OPT1_VAN_유 : BOOL; (* AT %MW15.8 *)
    HMI_M_차종수정_차종_OPT1_슬라이딩_무 : BOOL; (* AT %MW15.1 *)
    HMI_M_차종수정_차종_OPT1_슬라이딩_유 : BOOL; (* AT %MW15.0 *)
    HMI_M_차종수정_차종_OPT1_폴딩_무 : BOOL; (* AT %MW15.5 *)
    HMI_M_차종수정_차종_OPT1_폴딩_유 : BOOL; (* AT %MW15.4 *)
    HMI_M_차종수정_차종_공대차 : BOOL; (* AT %MW20.12 *)
    HMI_M_차종수정_차종_공차 : BOOL; (* AT %MW20.10 *)
    HMI_M_차종수정_차종_불량대차 : BOOL; (* AT %MW20.13 *)
    HMI_M_차종수정_차종_불량차 : BOOL; (* AT %MW20.11 *)
    HMI_M_차종수정가능_OK : BOOL; (* AT %MW9.4 *)
    HMI_M_차종수정가능_SEL : BOOL; (* AT %MW9.3 *)
    HMI_M_현재표출_차종 : ARRAY[0..19] OF WORD; (* AT %MW30 *)
    HMI_차종매칭_공정선택 : WORD; (* AT %MW8 *)
    HMI_차종수정_공정선택 : WORD; (* AT %MW7 *)
    ROOF_RACK_M_자동_운전중 : BOOL; (* AT %MW1500.4 *)
    ROOF_RACK_M_자동모드 : BOOL; (* AT %MW1500.1 *)
    S301_M_자동_운전중 : BOOL; (* S301 M 자동 운전중 *)
    S362_M_자동모드 : BOOL; (* AT %MW1000.1 *) (* S362 선택 자동모드 *)
    S364_M_자동모드 : BOOL; (* AT %MW2000.1 *) (* S364 선택 자동모드 *)
    S365_M_자동모드 : BOOL; (* AT %MW2500.1 *) (* S365 선택 자동모드 *)
    S366_M_자동_운전중 : BOOL; (* AT %MW3000.4 *) (* S366 자동운전중 *)
    S366_M_자동모드 : BOOL; (* AT %MW3000.1 *) (* S366 선택 자동모드 *)
    S367_M_자동모드 : BOOL; (* AT %MW3500.1 *) (* S367 선택 자동모드 *)
    S368_M_자동모드 : BOOL; (* AT %MW4000.1 *) (* S368 선택 자동모드 *)
    S369_1_M_자동모드 : BOOL; (* AT %MW4500.1 *) (* S369-1 선택 자동모드 *)
    S369_M_자동모드 : BOOL; (* AT %MW5000.1 *) (* S369 선택 자동모드 *)
END_VAR
VAR
    HMI_BT_MODIFY : FB470_HMI_BType_Modify_LS;
END_VAR
VAR
    _t1 : BOOL;
    _t2 : BOOL;
    _t3 : BOOL;
    _t4 : BOOL;
    _t5 : BOOL;
    _t6 : BOOL;
    _t7 : BOOL;
    _t8 : BOOL;
    _t9 : BOOL;
    _t10 : BOOL;
    _t11 : BOOL;
    _t12 : BOOL;
    _t13 : BOOL;
    _t14 : BOOL;
    _p15 : BOOL;
    _p16 : BOOL;
    _t17 : BOOL;
    _t18 : BOOL;
    _e19 : F_TRIG;
    _e20 : F_TRIG;
END_VAR

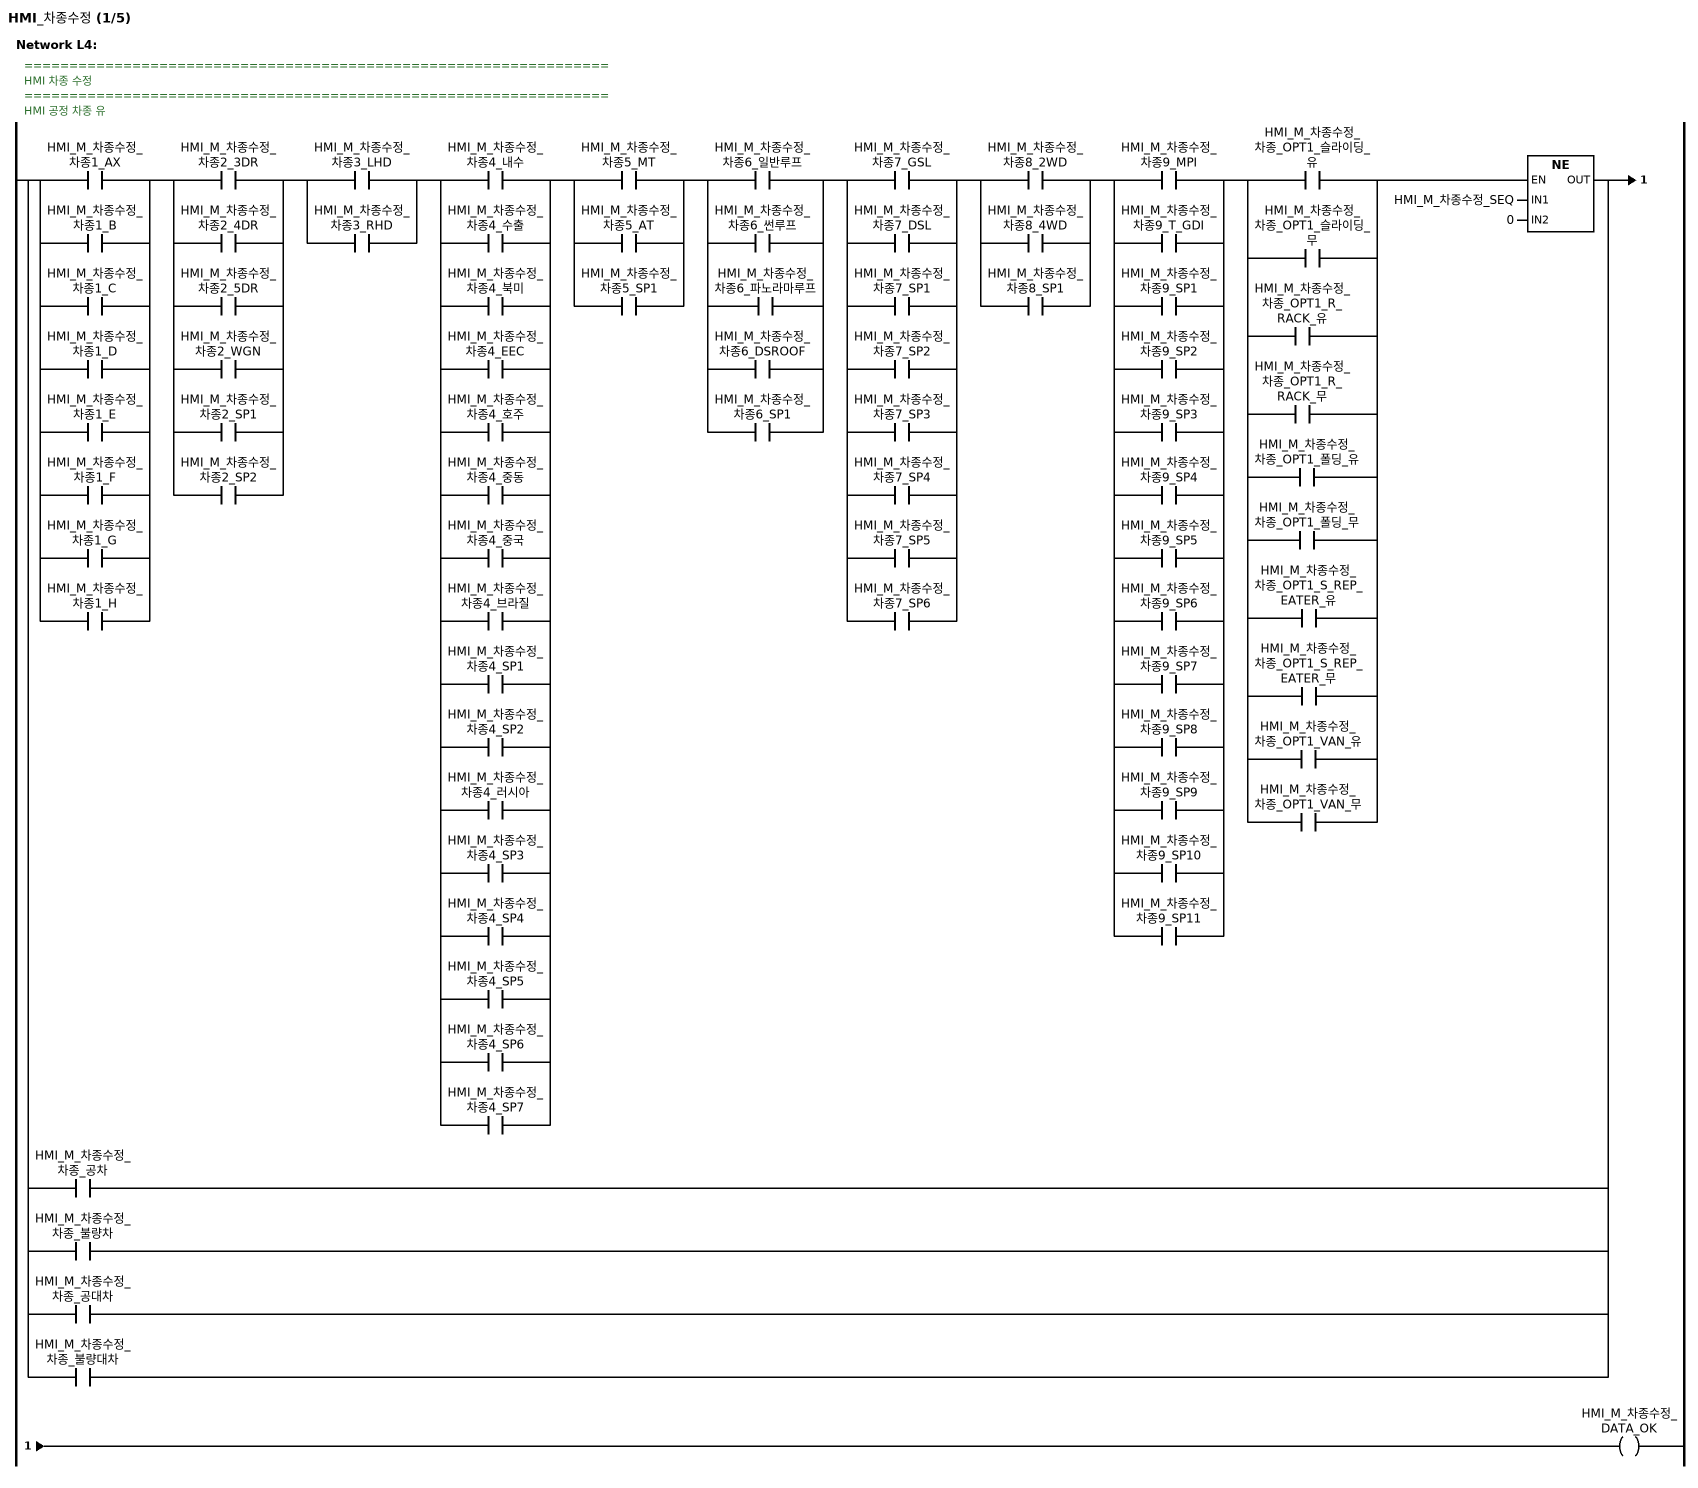
(* ================================================================= *)
(* HMI 차종 수정 *)
(* ================================================================= *)
(* HMI 공정 차종 유 *)
(* Rung L4 *)
IF (HMI_M_차종수정_차종1_AX OR HMI_M_차종수정_차종1_B OR HMI_M_차종수정_차종1_C OR HMI_M_차종수정_차종1_D OR HMI_M_차종수정_차종1_E OR HMI_M_차종수정_차종1_F OR HMI_M_차종수정_차종1_G OR HMI_M_차종수정_차종1_H) AND (HMI_M_차종수정_차종2_3DR OR HMI_M_차종수정_차종2_4DR OR HMI_M_차종수정_차종2_5DR OR HMI_M_차종수정_차종2_WGN OR HMI_M_차종수정_차종2_SP1 OR HMI_M_차종수정_차종2_SP2) AND (HMI_M_차종수정_차종3_LHD OR HMI_M_차종수정_차종3_RHD) AND (HMI_M_차종수정_차종4_내수 OR HMI_M_차종수정_차종4_수출 OR HMI_M_차종수정_차종4_북미 OR HMI_M_차종수정_차종4_EEC OR HMI_M_차종수정_차종4_호주 OR HMI_M_차종수정_차종4_중동 OR HMI_M_차종수정_차종4_중국 OR HMI_M_차종수정_차종4_브라질 OR HMI_M_차종수정_차종4_SP1 OR HMI_M_차종수정_차종4_SP2 OR HMI_M_차종수정_차종4_러시아 OR HMI_M_차종수정_차종4_SP3 OR HMI_M_차종수정_차종4_SP4 OR HMI_M_차종수정_차종4_SP5 OR HMI_M_차종수정_차종4_SP6 OR HMI_M_차종수정_차종4_SP7) AND (HMI_M_차종수정_차종5_MT OR HMI_M_차종수정_차종5_AT OR HMI_M_차종수정_차종5_SP1) AND (HMI_M_차종수정_차종6_일반루프 OR HMI_M_차종수정_차종6_썬루프 OR HMI_M_차종수정_차종6_파노라마루프 OR HMI_M_차종수정_차종6_DSROOF OR HMI_M_차종수정_차종6_SP1) AND (HMI_M_차종수정_차종7_GSL OR HMI_M_차종수정_차종7_DSL OR HMI_M_차종수정_차종7_SP1 OR HMI_M_차종수정_차종7_SP2 OR HMI_M_차종수정_차종7_SP3 OR HMI_M_차종수정_차종7_SP4 OR HMI_M_차종수정_차종7_SP5 OR HMI_M_차종수정_차종7_SP6) AND (HMI_M_차종수정_차종8_2WD OR HMI_M_차종수정_차종8_4WD OR HMI_M_차종수정_차종8_SP1) AND (HMI_M_차종수정_차종9_MPI OR HMI_M_차종수정_차종9_T_GDI OR HMI_M_차종수정_차종9_SP1 OR HMI_M_차종수정_차종9_SP2 OR HMI_M_차종수정_차종9_SP3 OR HMI_M_차종수정_차종9_SP4 OR HMI_M_차종수정_차종9_SP5 OR HMI_M_차종수정_차종9_SP6 OR HMI_M_차종수정_차종9_SP7 OR HMI_M_차종수정_차종9_SP8 OR HMI_M_차종수정_차종9_SP9 OR HMI_M_차종수정_차종9_SP10 OR HMI_M_차종수정_차종9_SP11) AND (HMI_M_차종수정_차종_OPT1_슬라이딩_유 OR HMI_M_차종수정_차종_OPT1_슬라이딩_무 OR HMI_M_차종수정_차종_OPT1_R_RACK_유 OR HMI_M_차종수정_차종_OPT1_R_RACK_무 OR HMI_M_차종수정_차종_OPT1_폴딩_유 OR HMI_M_차종수정_차종_OPT1_폴딩_무 OR HMI_M_차종수정_차종_OPT1_S_REP_EATER_유 OR HMI_M_차종수정_차종_OPT1_S_REP_EATER_무 OR HMI_M_차종수정_차종_OPT1_VAN_유 OR HMI_M_차종수정_차종_OPT1_VAN_무) THEN
    _t1 := HMI_M_차종수정_SEQ <> 0;
END_IF;
HMI_M_차종수정_DATA_OK := _t1 OR HMI_M_차종수정_차종_공차 OR HMI_M_차종수정_차종_불량차 OR HMI_M_차종수정_차종_공대차 OR HMI_M_차종수정_차종_불량대차;

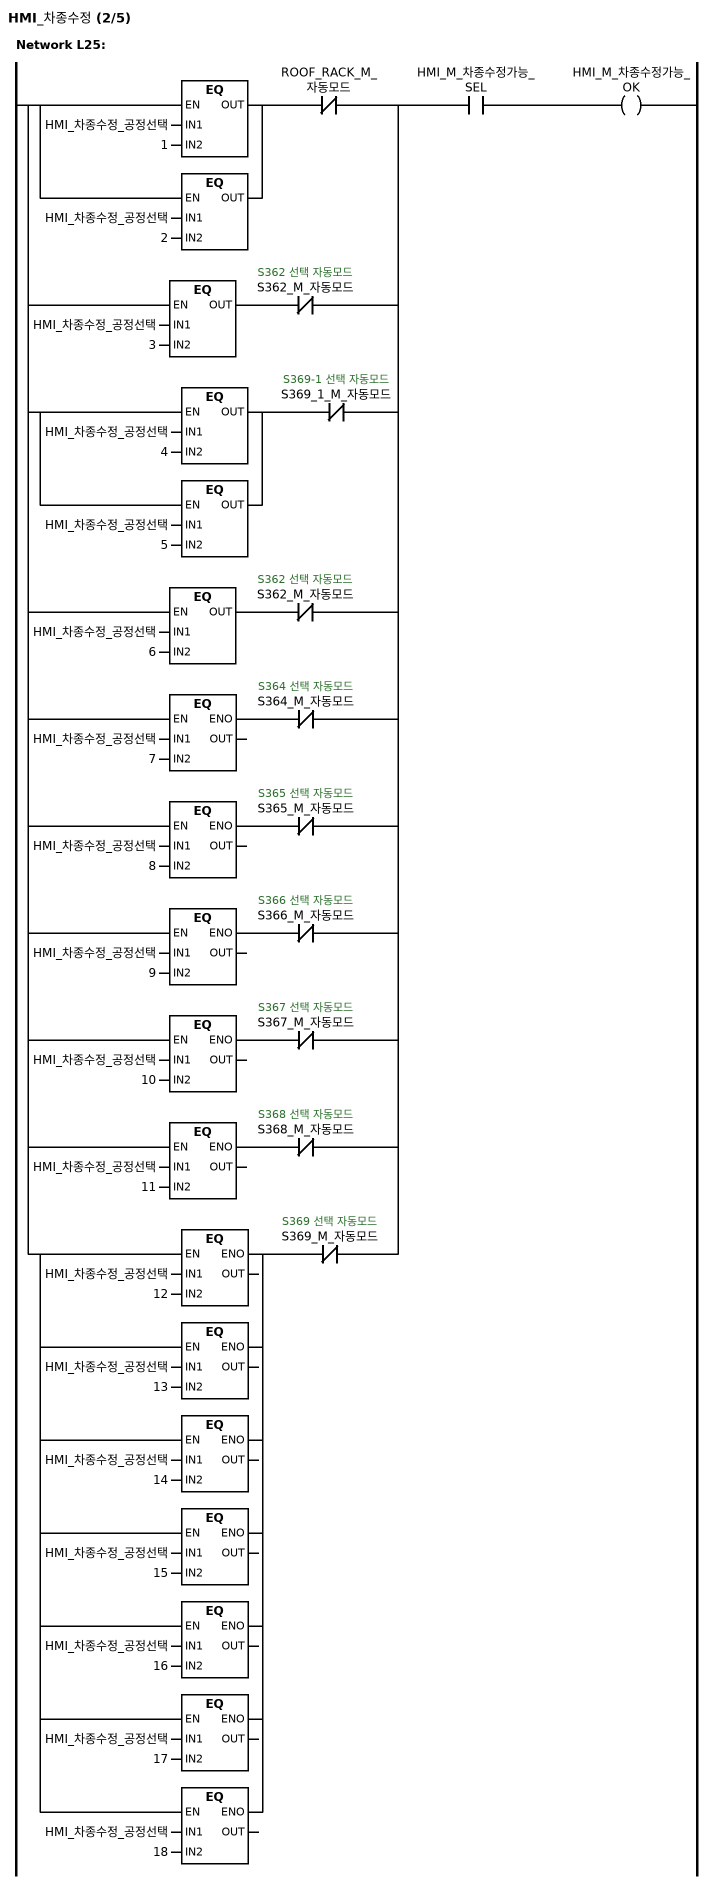
(* Rung L25 *)
_t2 := HMI_차종수정_공정선택 = 7;
_t3 := HMI_차종수정_공정선택 = 8;
_t4 := HMI_차종수정_공정선택 = 9;
_t5 := HMI_차종수정_공정선택 = 10;
_t6 := HMI_차종수정_공정선택 = 11;
_t7 := HMI_차종수정_공정선택 = 12;
_t8 := HMI_차종수정_공정선택 = 13;
_t9 := HMI_차종수정_공정선택 = 14;
_t10 := HMI_차종수정_공정선택 = 15;
_t11 := HMI_차종수정_공정선택 = 16;
_t12 := HMI_차종수정_공정선택 = 17;
_t13 := HMI_차종수정_공정선택 = 18;
HMI_M_차종수정가능_OK := ((((HMI_차종수정_공정선택 = 1) OR (HMI_차종수정_공정선택 = 2)) AND NOT ROOF_RACK_M_자동모드) OR ((HMI_차종수정_공정선택 = 3) AND NOT S362_M_자동모드) OR (((HMI_차종수정_공정선택 = 4) OR (HMI_차종수정_공정선택 = 5)) AND NOT S369_1_M_자동모드) OR ((HMI_차종수정_공정선택 = 6) AND NOT S362_M_자동모드) OR NOT S364_M_자동모드 OR NOT S365_M_자동모드 OR NOT S366_M_자동모드 OR NOT S367_M_자동모드 OR NOT S368_M_자동모드 OR NOT S369_M_자동모드) AND HMI_M_차종수정가능_SEL;

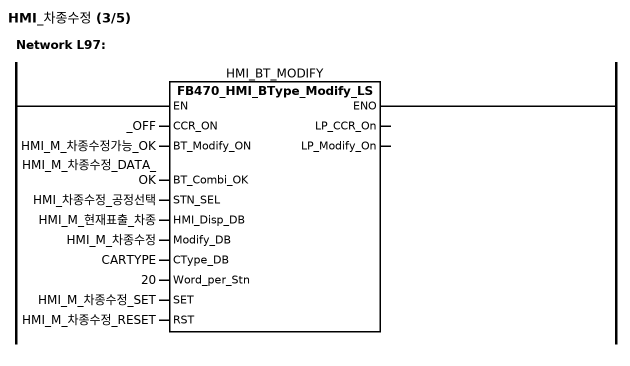
(* Rung L97 *)
HMI_BT_MODIFY(CCR_ON := _OFF, BT_Modify_ON := HMI_M_차종수정가능_OK, BT_Combi_OK := HMI_M_차종수정_DATA_OK, STN_SEL := HMI_차종수정_공정선택, HMI_Disp_DB := HMI_M_현재표출_차종, Modify_DB := HMI_M_차종수정, CType_DB := CARTYPE, Word_per_Stn := 20, SET := HMI_M_차종수정_SET, RST := HMI_M_차종수정_RESET);

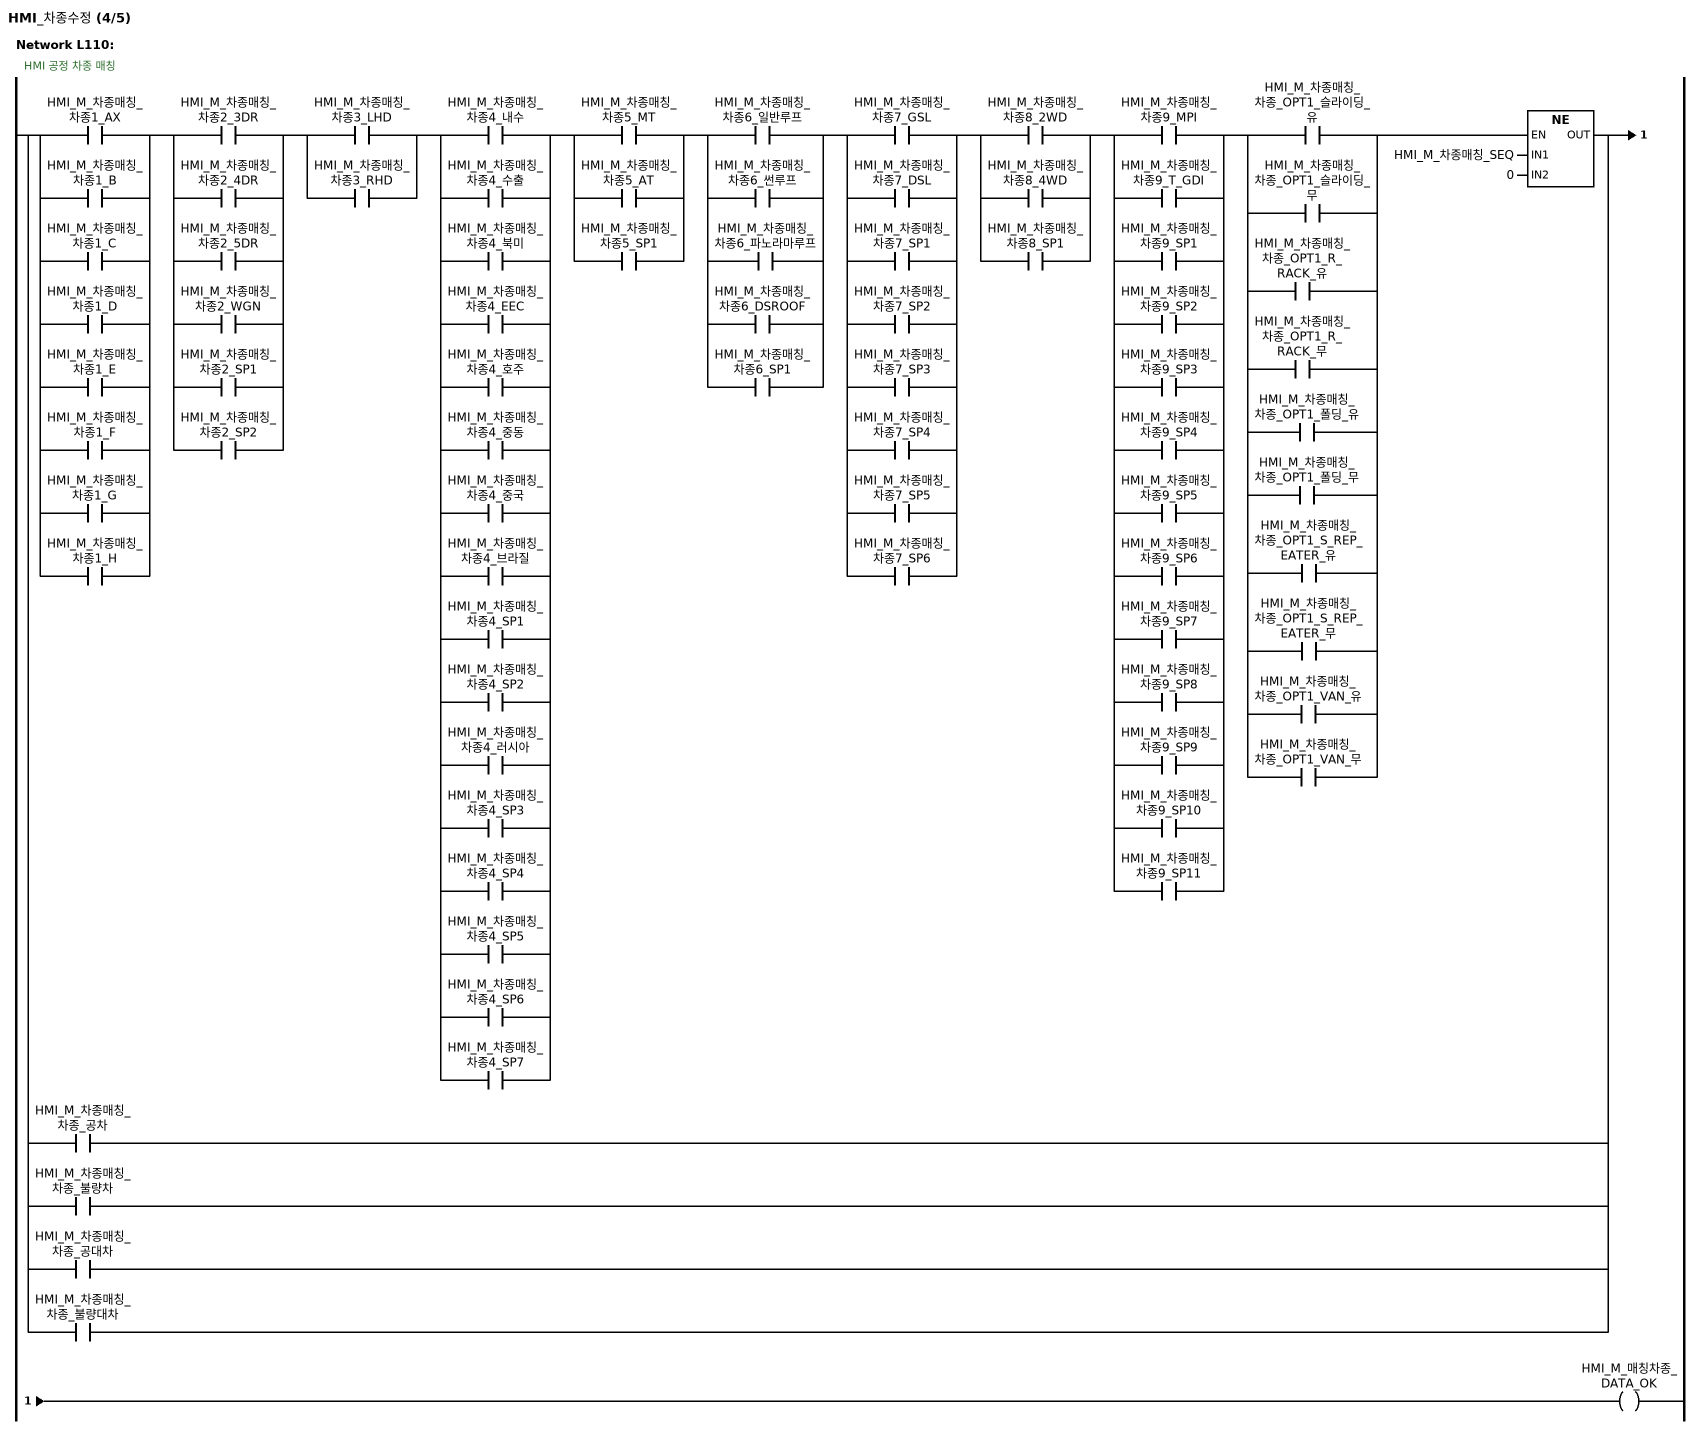
(* HMI 공정 차종 매칭 *)
(* Rung L110 *)
IF (HMI_M_차종매칭_차종1_AX OR HMI_M_차종매칭_차종1_B OR HMI_M_차종매칭_차종1_C OR HMI_M_차종매칭_차종1_D OR HMI_M_차종매칭_차종1_E OR HMI_M_차종매칭_차종1_F OR HMI_M_차종매칭_차종1_G OR HMI_M_차종매칭_차종1_H) AND (HMI_M_차종매칭_차종2_3DR OR HMI_M_차종매칭_차종2_4DR OR HMI_M_차종매칭_차종2_5DR OR HMI_M_차종매칭_차종2_WGN OR HMI_M_차종매칭_차종2_SP1 OR HMI_M_차종매칭_차종2_SP2) AND (HMI_M_차종매칭_차종3_LHD OR HMI_M_차종매칭_차종3_RHD) AND (HMI_M_차종매칭_차종4_내수 OR HMI_M_차종매칭_차종4_수출 OR HMI_M_차종매칭_차종4_북미 OR HMI_M_차종매칭_차종4_EEC OR HMI_M_차종매칭_차종4_호주 OR HMI_M_차종매칭_차종4_중동 OR HMI_M_차종매칭_차종4_중국 OR HMI_M_차종매칭_차종4_브라질 OR HMI_M_차종매칭_차종4_SP1 OR HMI_M_차종매칭_차종4_SP2 OR HMI_M_차종매칭_차종4_러시아 OR HMI_M_차종매칭_차종4_SP3 OR HMI_M_차종매칭_차종4_SP4 OR HMI_M_차종매칭_차종4_SP5 OR HMI_M_차종매칭_차종4_SP6 OR HMI_M_차종매칭_차종4_SP7) AND (HMI_M_차종매칭_차종5_MT OR HMI_M_차종매칭_차종5_AT OR HMI_M_차종매칭_차종5_SP1) AND (HMI_M_차종매칭_차종6_일반루프 OR HMI_M_차종매칭_차종6_썬루프 OR HMI_M_차종매칭_차종6_파노라마루프 OR HMI_M_차종매칭_차종6_DSROOF OR HMI_M_차종매칭_차종6_SP1) AND (HMI_M_차종매칭_차종7_GSL OR HMI_M_차종매칭_차종7_DSL OR HMI_M_차종매칭_차종7_SP1 OR HMI_M_차종매칭_차종7_SP2 OR HMI_M_차종매칭_차종7_SP3 OR HMI_M_차종매칭_차종7_SP4 OR HMI_M_차종매칭_차종7_SP5 OR HMI_M_차종매칭_차종7_SP6) AND (HMI_M_차종매칭_차종8_2WD OR HMI_M_차종매칭_차종8_4WD OR HMI_M_차종매칭_차종8_SP1) AND (HMI_M_차종매칭_차종9_MPI OR HMI_M_차종매칭_차종9_T_GDI OR HMI_M_차종매칭_차종9_SP1 OR HMI_M_차종매칭_차종9_SP2 OR HMI_M_차종매칭_차종9_SP3 OR HMI_M_차종매칭_차종9_SP4 OR HMI_M_차종매칭_차종9_SP5 OR HMI_M_차종매칭_차종9_SP6 OR HMI_M_차종매칭_차종9_SP7 OR HMI_M_차종매칭_차종9_SP8 OR HMI_M_차종매칭_차종9_SP9 OR HMI_M_차종매칭_차종9_SP10 OR HMI_M_차종매칭_차종9_SP11) AND (HMI_M_차종매칭_차종_OPT1_슬라이딩_유 OR HMI_M_차종매칭_차종_OPT1_슬라이딩_무 OR HMI_M_차종매칭_차종_OPT1_R_RACK_유 OR HMI_M_차종매칭_차종_OPT1_R_RACK_무 OR HMI_M_차종매칭_차종_OPT1_폴딩_유 OR HMI_M_차종매칭_차종_OPT1_폴딩_무 OR HMI_M_차종매칭_차종_OPT1_S_REP_EATER_유 OR HMI_M_차종매칭_차종_OPT1_S_REP_EATER_무 OR HMI_M_차종매칭_차종_OPT1_VAN_유 OR HMI_M_차종매칭_차종_OPT1_VAN_무) THEN
    _t14 := HMI_M_차종매칭_SEQ <> 0;
END_IF;
HMI_M_매칭차종_DATA_OK := _t14 OR HMI_M_차종매칭_차종_공차 OR HMI_M_차종매칭_차종_불량차 OR HMI_M_차종매칭_차종_공대차 OR HMI_M_차종매칭_차종_불량대차;

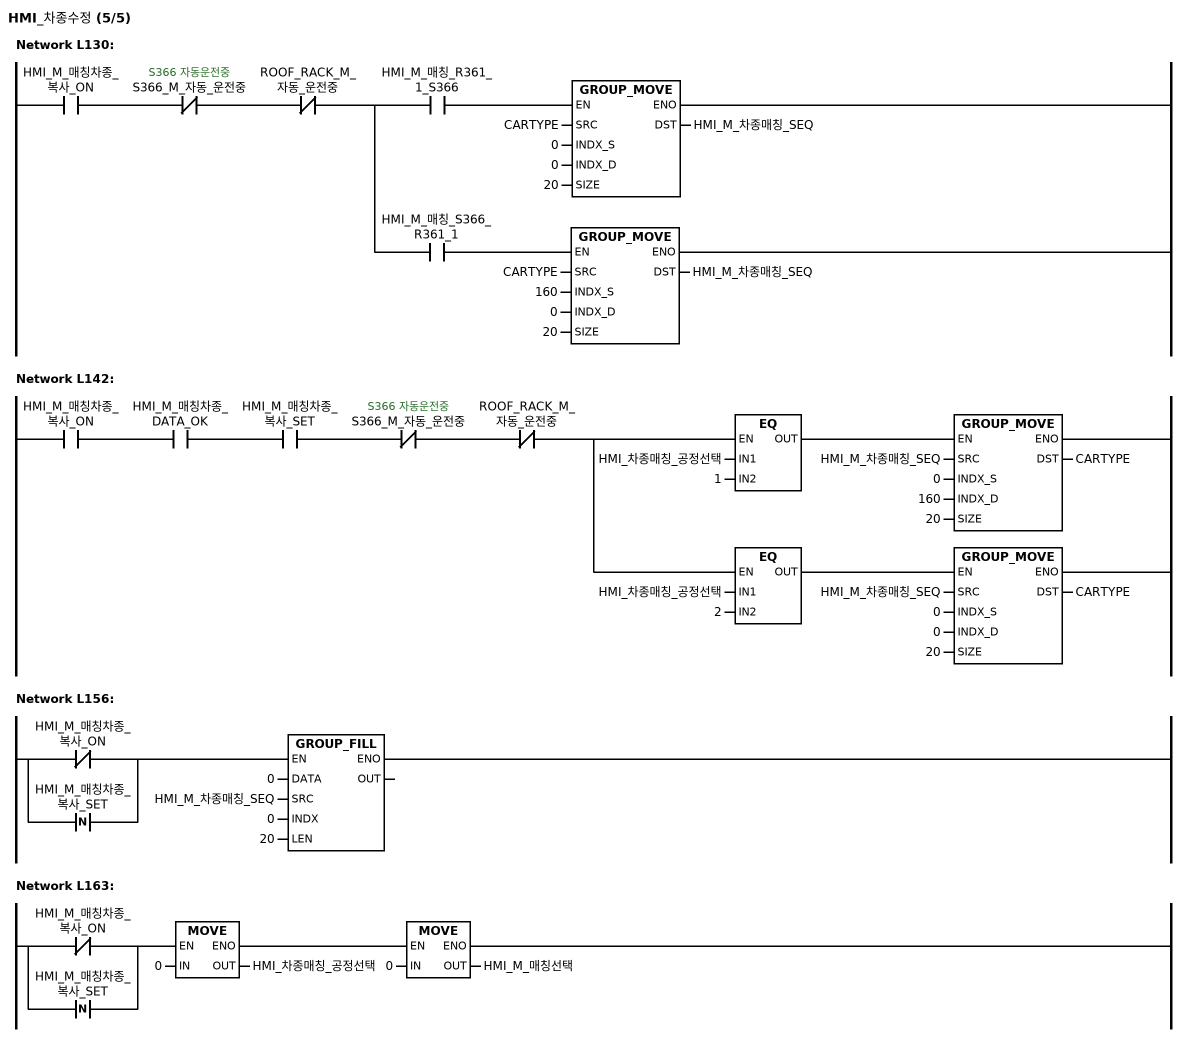
(* Rung L130 *)
_p15 := HMI_M_매칭차종_복사_ON AND NOT S366_M_자동_운전중 AND NOT ROOF_RACK_M_자동_운전중;
IF _p15 AND HMI_M_매칭_R361_1_S366 THEN
    HMI_M_차종매칭_SEQ := GROUP_MOVE(SRC := CARTYPE, INDX_S := 0, INDX_D := 0, SIZE := 20);
END_IF;
IF _p15 AND HMI_M_매칭_S366_R361_1 THEN
    HMI_M_차종매칭_SEQ := GROUP_MOVE(SRC := CARTYPE, INDX_S := 160, INDX_D := 0, SIZE := 20);
END_IF;
(* Rung L142 *)
_p16 := HMI_M_매칭차종_복사_ON AND HMI_M_매칭차종_DATA_OK AND HMI_M_매칭차종_복사_SET AND NOT S366_M_자동_운전중 AND NOT ROOF_RACK_M_자동_운전중;
IF _p16 THEN _t17 := HMI_차종매칭_공정선택 = 1; END_IF;
IF _t17 THEN CARTYPE := GROUP_MOVE(SRC := HMI_M_차종매칭_SEQ, INDX_S := 0, INDX_D := 160, SIZE := 20); END_IF;
IF _p16 THEN _t18 := HMI_차종매칭_공정선택 = 2; END_IF;
IF _t18 THEN CARTYPE := GROUP_MOVE(SRC := HMI_M_차종매칭_SEQ, INDX_S := 0, INDX_D := 0, SIZE := 20); END_IF;
(* Rung L156 *)
_e19(CLK := HMI_M_매칭차종_복사_SET);
IF NOT HMI_M_매칭차종_복사_ON OR _e19.Q THEN
    GROUP_FILL(DATA := 0, SRC := HMI_M_차종매칭_SEQ, INDX := 0, LEN := 20);
END_IF;
(* Rung L163 *)
_e20(CLK := HMI_M_매칭차종_복사_SET);
IF NOT HMI_M_매칭차종_복사_ON OR _e20.Q THEN
    HMI_차종매칭_공정선택 := 0;
    HMI_M_매칭선택 := 0;
END_IF;
END_PROGRAM

PROGRAM 차종전송 (* task: 스캔 프로그램 *)
VAR_EXTERNAL RETAIN
    CARTYPE : ARRAY[0..599] OF WORD; (* AT %MW10000 *) (* CARTYPE *)
    R361_1_M_DATA_삭제_PLS : BOOL; (* AT %MW9000.0 *) (* R361 1 M DATA 삭제 PLS *)
    R361_1_M_DATA_삭제_완료 : BOOL; (* AT %MW9000.2 *) (* R361 1 M DATA 삭제 완료 *)
    R361_1_M_S365_DATA_전송_MEMO : BOOL; (* AT %MW9000.4 *) (* R361 1 M S365 DATA 전송 MEMO *)
    R361_1_M_S365_DATA_전송_PLS : BOOL; (* AT %MW9000.5 *) (* R361 1 M S365 DATA 전송 PLS *)
    R361_1_M_차종_무 : BOOL; (* AT %MW1502.1 *)
    R361_1_M_차종_유 : BOOL; (* AT %MW1502.0 *)
    R361_2_M_DATA_삭제_PLS : BOOL; (* AT %MW9001.0 *) (* R361 2 M DATA 삭제 PLS *)
    R361_2_M_DATA_삭제_완료 : BOOL; (* AT %MW9001.2 *) (* R361 2 M DATA 삭제 완료 *)
    R361_2_M_R361_1_DATA_전송_MEMO : BOOL; (* AT %MW9001.8 *) (* R361 2 M R361 1 DATA 전송 MEMO *)
    R361_2_M_R361_1_DATA_전송_PLS : BOOL; (* AT %MW9001.9 *) (* R361 2 M R361 1 DATA 전송 PLS *)
    R361_2_M_R361_1_DATA_전송_완료 : BOOL; (* AT %MW9001.11 *) (* R361 2 M R361 1 DATA 전송 완료 *)
    R361_2_M_S364_DATA_전송_MEMO : BOOL; (* AT %MW9001.4 *) (* R361 2 M S364 DATA 전송 MEMO *)
    R361_2_M_S364_DATA_전송_PLS : BOOL; (* AT %MW9001.5 *) (* R361 2 M S364 DATA 전송 PLS *)
    R361_2_M_차종_OPT1_R_RACK_무 : BOOL; (* AT %MW10025.3 *) (* R361 2 M 차종 OPT1 R RACK 무 *)
    R361_2_M_차종_유 : BOOL; (* AT %MW1502.2 *)
    R363_2_M_S366_DATA_전송_MEMO : BOOL; (* AT %MW9003.8 *) (* R363_2 M S366 DATA 전송 MEMO *)
    R363_2_M_S366_DATA_전송_PLS : BOOL; (* AT %MW9003.9 *) (* R363_2 M S366 DATA 전송 PLS *)
    R363_2_M_S366_DATA_전송_완료 : BOOL; (* AT %MW9003.11 *) (* R363_2 M S366 DATA 전송 완료 *)
    R363_2_M_차종_무 : BOOL; (* AT %MW1002.3 *)
    R363_2_M_차종_유 : BOOL; (* AT %MW1002.2 *) (* S362_M_공정_차종_보조 *)
    R369_1_M_S368_DATA_전송_MEMO : BOOL; (* AT %MW9007.4 *) (* R369 1 M S368 DATA 전송 MEMO *)
    R369_1_M_S368_DATA_전송_PLS : BOOL; (* AT %MW9007.5 *) (* R369 1 M S368 DATA 전송 PLS *)
    R369_1_M_S369_1_DATA_전송_MEMO : BOOL; (* AT %MW9007.8 *) (* R369 1 M S369 1 DATA 전송 MEMO *)
    R369_1_M_S369_1_DATA_전송_PLS : BOOL; (* AT %MW9007.9 *) (* R369 1 M S369 1 DATA 전송 PLS *)
    R369_1_M_S369_1_DATA_전송_완료 : BOOL; (* AT %MW9007.11 *) (* R369 1 M S369 1 DATA 전송 완료 *)
    R369_1_M_차종_무 : BOOL; (* AT %MW4502.3 *)
    R369_1_M_차종_유 : BOOL; (* AT %MW4502.2 *)
    R369_2_M_로딩버퍼_DATA_전송_MEMO : BOOL; (* AT %MW9008.8 *) (* R369 2 M 로딩버퍼 DATA 전송 MEMO *)
    R369_2_M_로딩버퍼_DATA_전송_PLS : BOOL; (* AT %MW9008.9 *) (* R369 2 M 로딩버퍼 DATA 전송 PLS *)
    R369_2_M_로딩버퍼_DATA_전송_완료 : BOOL; (* AT %MW9008.11 *) (* R369 2 M 로딩버퍼 DATA 전송 완료 *)
    R369_2_M_차종_무 : BOOL; (* AT %MW4502.5 *)
    R369_2_M_차종_유 : BOOL; (* AT %MW4502.4 *)
    S362_M_R363_2_DATA_전송_MEMO : BOOL; (* AT %MW9010.4 *) (* S362 M R363 2 DATA 전송 MEMO *)
    S362_M_R363_2_DATA_전송_PLS : BOOL; (* AT %MW9010.5 *) (* S362 M R363 2 DATA 전송 PLS *)
    S362_M_R363_2_DATA_전송_완료 : BOOL; (* AT %MW9010.7 *) (* S362 M R363 2 DATA 전송 완료 *)
    S362_M_R363_2_언로딩_완료 : BOOL; (* AT %MW1001.3 *)
    S362_M_공정_차종_유 : BOOL; (* AT %MW1002.0 *) (* S362_M_공정_차종_유 *)
    S364_M_DATA_삭제_PLS : BOOL; (* AT %MW9012.0 *) (* S364 M DATA 삭제 PLS *)
    S364_M_DATA_삭제_완료 : BOOL; (* AT %MW9012.2 *) (* S364 M DATA 삭제 완료 *)
    S364_M_R361_1_언로딩완료 : BOOL; (* AT %MW2001.4 *)
    S364_M_공정_제품감지_무 : BOOL; (* AT %MW2002.5 *) (* S364_M_공정_제품감지_무 *)
    S364_M_공정_차종_무 : BOOL; (* AT %MW2002.1 *) (* S364_M_공정_차종_무 *)
    S364_M_공정_차종_유 : BOOL; (* AT %MW2002.0 *) (* S364_M_공정_차종_유 *)
    S365_M_DATA_삭제_PLS : BOOL; (* AT %MW9013.0 *) (* S365 M DATA 삭제 PLS *)
    S365_M_DATA_삭제_완료 : BOOL; (* AT %MW9013.2 *) (* S365 M DATA 삭제 완료 *)
    S365_M_R361_1_안착완료 : BOOL; (* AT %MW2501.1 *)
    S365_M_R361_1_언로딩완료 : BOOL; (* AT %MW2501.2 *)
    S365_M_공정_제품감지_무 : BOOL; (* AT %MW2501.4 *) (* S365_M_공정_제품감지_무 *)
    S365_M_공정_차종_무 : BOOL; (* AT %MW2502.1 *) (* S365_M_공정_차종_무 *)
    S365_M_공정_차종_유 : BOOL; (* AT %MW2502.0 *) (* S365_M_공정_차종_유 *)
    S366_M_DATA_삭제_PLS : BOOL; (* AT %MW9014.0 *) (* S366 M DATA 삭제 PLS *)
    S366_M_DATA_삭제_완료 : BOOL; (* AT %MW9014.2 *) (* S366 M DATA 삭제 완료 *)
    S366_M_R361_1_ROOF_로딩완료 : BOOL; (* AT %MW3001.2 *)
    S366_M_R361_1_언로딩완료 : BOOL; (* AT %MW3001.4 *)
    S366_M_R363_2_RAIL_로딩완료 : BOOL; (* AT %MW3001.1 *)
    S366_M_공정_제품감지_무 : BOOL; (* AT %MW3001.7 *) (* S366_M_공정_제품감지_무 *)
    S366_M_공정_차종_무 : BOOL; (* AT %MW3002.1 *) (* S366_M_공정_차종_무 *)
    S366_M_공정_차종_유 : BOOL; (* AT %MW3002.0 *) (* S366_M_공정_차종_유 *)
    S367_M_DATA_삭제_PLS : BOOL; (* AT %MW9015.0 *) (* S367 M DATA 삭제 PLS *)
    S367_M_DATA_삭제_완료 : BOOL; (* AT %MW9015.2 *) (* S367 M DATA 삭제 완료 *)
    S367_M_R369_1_DATA_전송_MEMO : BOOL; (* AT %MW9015.8 *) (* S367 M R369 1 DATA 전송 MEMO *)
    S367_M_R369_1_DATA_전송_PLS : BOOL; (* AT %MW9015.9 *) (* S367 M R369 1 DATA 전송 PLS *)
    S367_M_R369_1_DATA_전송_완료 : BOOL; (* AT %MW9015.11 *) (* S367 M R369 1 DATA 전송 완료 *)
    S367_M_R369_1_언로딩완료 : BOOL; (* AT %MW3501.3 *)
    S367_M_공정_제품감지_무 : BOOL; (* AT %MW3501.6 *) (* S367_M_공정_제품감지_무 *)
    S367_M_공정_차종_유 : BOOL; (* AT %MW3502.0 *) (* S367_M_공정_차종_유 *)
    S368_M_DATA_삭제_PLS : BOOL; (* AT %MW9016.0 *) (* S368 M DATA 삭제 PLS *)
    S368_M_DATA_삭제_완료 : BOOL; (* AT %MW9016.2 *) (* S368 M DATA 삭제 완료 *)
    S368_M_R369_1_안착완료 : BOOL; (* AT %MW4001.1 *)
    S368_M_R369_1_언로딩완료 : BOOL; (* AT %MW4001.4 *)
    S368_M_공정_제품감지_무 : BOOL; (* AT %MW4001.6 *) (* S368_M_공정_제품감지_무 *)
    S368_M_공정_차종_무 : BOOL; (* AT %MW4002.1 *) (* S368_M_공정_차종_무 *)
    S368_M_공정_차종_유 : BOOL; (* AT %MW4002.0 *) (* S368_M_공정_차종_유 *)
    S369_1_M_R369_1_안착완료 : BOOL; (* AT %MW4501.1 *)
    S369_1_M_R369_2_DATA_전송_MEMO : BOOL; (* AT %MW9018.8 *) (* S369_1 M R369 2 DATA 전송 MEMO *)
    S369_1_M_R369_2_DATA_전송_PLS : BOOL; (* AT %MW9018.9 *) (* S369_1 M R369 2 DATA 전송 PLS *)
    S369_1_M_R369_2_DATA_전송_완료 : BOOL; (* AT %MW9018.11 *) (* S369_1 M R369 2 DATA 전송 완료 *)
    S369_1_M_R369_2_언로딩완료 : BOOL; (* AT %MW4501.2 *)
    S369_1_M_공정_차종_무 : BOOL; (* AT %MW4502.1 *) (* S369_1_M_공정_차종_무 *)
    S369_1_M_공정_차종_유 : BOOL; (* AT %MW4502.0 *) (* S369_1_M_공정_차종_유 *)
    S369_M_R308_3_언로딩완료 : BOOL; (* AT %MW5001.5 *)
    S369_M_R369_2_로딩완료 : BOOL; (* AT %MW5001.2 *)
    S369_M_로딩_리셋보조 : BOOL; (* AT %MW5000.13 *)
    S369_M_로딩버퍼_차종_무 : BOOL; (* AT %MW5002.1 *)
    S369_M_로딩버퍼_차종_유 : BOOL; (* AT %MW5002.0 *)
    S369_M_언로딩_이젝터_제품감지_무 : BOOL; (* AT %MW5001.11 *)
    S369_M_전체_컨베어_도착완료 : BOOL; (* AT %MW5003.0 *)
    S369_언로딩버퍼_M_DATA_삭제_PLS : BOOL; (* AT %MW9021.0 *) (* S369_언로딩버퍼 M DATA 삭제 PLS *)
    S369_언로딩버퍼_M_DATA_삭제_완료 : BOOL; (* AT %MW9021.2 *) (* S369_언로딩버퍼 M DATA 삭제 완료 *)
    S369_컨베어_M_DATA_전송_MEMO : BOOL; (* AT %MW9020.8 *) (* S369_컨베어 M 이송버퍼02 DATA 전송 MEMO *)
    S369_컨베어_M_DATA_전송_PLS : BOOL; (* AT %MW9020.9 *) (* S369_컨베어 M 이송버퍼02 DATA 전송 PLS *)
    S369_컨베어_M_DATA_전송_완료 : BOOL; (* AT %MW9020.11 *) (* S369_컨베어 M 이송버퍼02 DATA 전송 완료 *)
END_VAR
VAR
    INST : FB409_Car_Type_Clear_v1;
    INST1 : FB409_Car_Type_Clear_v1;
    INST10 : FB407_Car_Type_Move_Stn_v1;
    INST11 : FB409_Car_Type_Clear_v1;
    INST12 : FB407_Car_Type_Move_Stn_v1;
    INST13 : FB407_Car_Type_Move_Stn_v1;
    INST14 : FB407_Car_Type_Move_Stn_v1;
    INST15 : FB409_Car_Type_Clear_v1;
    INST16 : FB407_Car_Type_Move_Stn_v1;
    INST17 : FB407_Car_Type_Move_Stn_v1;
    INST18 : FB409_Car_Type_Clear_v1;
    INST19 : FB406_Car_Type_Move_Line_v1;
    INST2 : FB409_Car_Type_Clear_v1;
    INST3 : FB409_Car_Type_Clear_v1;
    INST4 : FB409_Car_Type_Clear_v1;
    INST5 : FB409_Car_Type_Clear_v1;
    INST6 : FB407_Car_Type_Move_Stn_v1;
    INST7 : FB409_Car_Type_Clear_v1;
    INST8 : FB409_Car_Type_Clear_v1;
    INST9 : FB407_Car_Type_Move_Stn_v1;
END_VAR
VAR_EXTERNAL
    R361_1_M_I_RB_2차_작업완료 : BOOL; (* AT %MW20011.3 *) (* R361_1_M_I_RB_2차_작업완료 *)
    R361_1_M_I_RB_최종작업완료 : BOOL; (* AT %MW20011.0 *) (* R361_1_M_I_RB_최종작업완료 *)
    R361_2_M_I_RB_2차_작업완료 : BOOL; (* AT %MW20021.3 *) (* R361_2_M_I_RB_2차_작업완료 *)
    R361_2_M_I_RB_최종작업완료 : BOOL; (* AT %MW20021.0 *) (* R361_2_M_I_RB_최종작업완료 *)
END_VAR

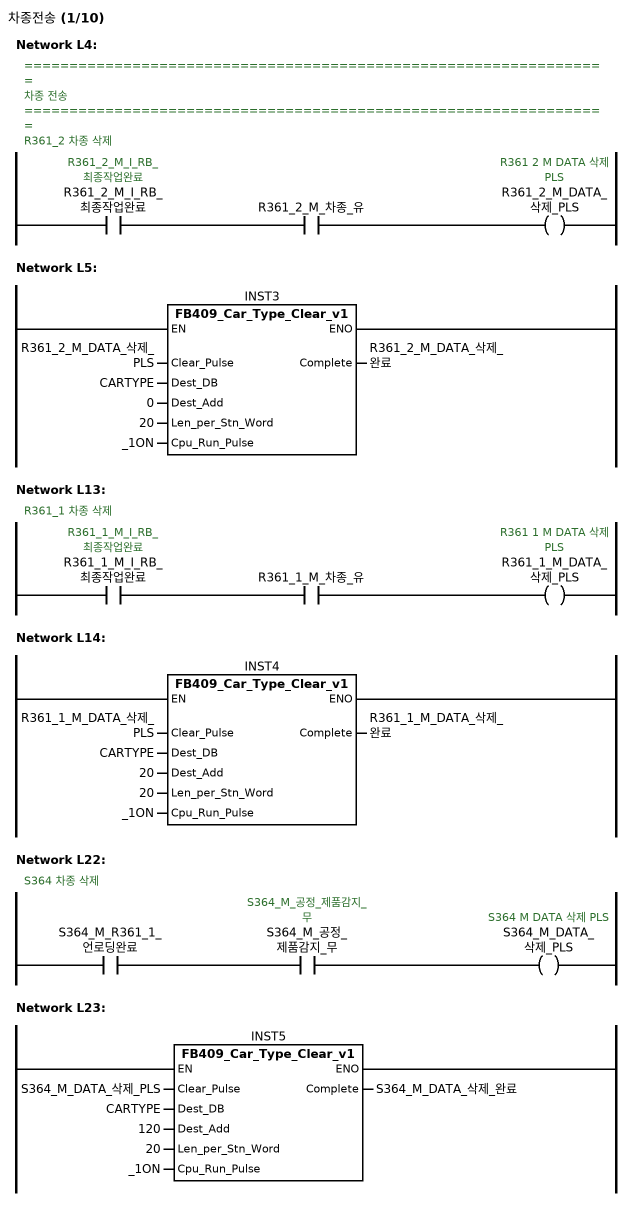
(* ================================================================= *)
(* 차종 전송 *)
(* ================================================================= *)
(* R361_2 차종 삭제 *)
(* Rung L4 *)
R361_2_M_DATA_삭제_PLS := R361_2_M_I_RB_최종작업완료 AND R361_2_M_차종_유;
(* Rung L5 *)
INST3(Clear_Pulse := R361_2_M_DATA_삭제_PLS, Dest_DB := CARTYPE, Dest_Add := 0, Len_per_Stn_Word := 20, Cpu_Run_Pulse := _1ON, Complete => R361_2_M_DATA_삭제_완료);
(* R361_1 차종 삭제 *)
(* Rung L13 *)
R361_1_M_DATA_삭제_PLS := R361_1_M_I_RB_최종작업완료 AND R361_1_M_차종_유;
(* Rung L14 *)
INST4(Clear_Pulse := R361_1_M_DATA_삭제_PLS, Dest_DB := CARTYPE, Dest_Add := 20, Len_per_Stn_Word := 20, Cpu_Run_Pulse := _1ON, Complete => R361_1_M_DATA_삭제_완료);
(* S364 차종 삭제 *)
(* Rung L22 *)
S364_M_DATA_삭제_PLS := S364_M_R361_1_언로딩완료 AND S364_M_공정_제품감지_무;
(* Rung L23 *)
INST5(Clear_Pulse := S364_M_DATA_삭제_PLS, Dest_DB := CARTYPE, Dest_Add := 120, Len_per_Stn_Word := 20, Cpu_Run_Pulse := _1ON, Complete => S364_M_DATA_삭제_완료);

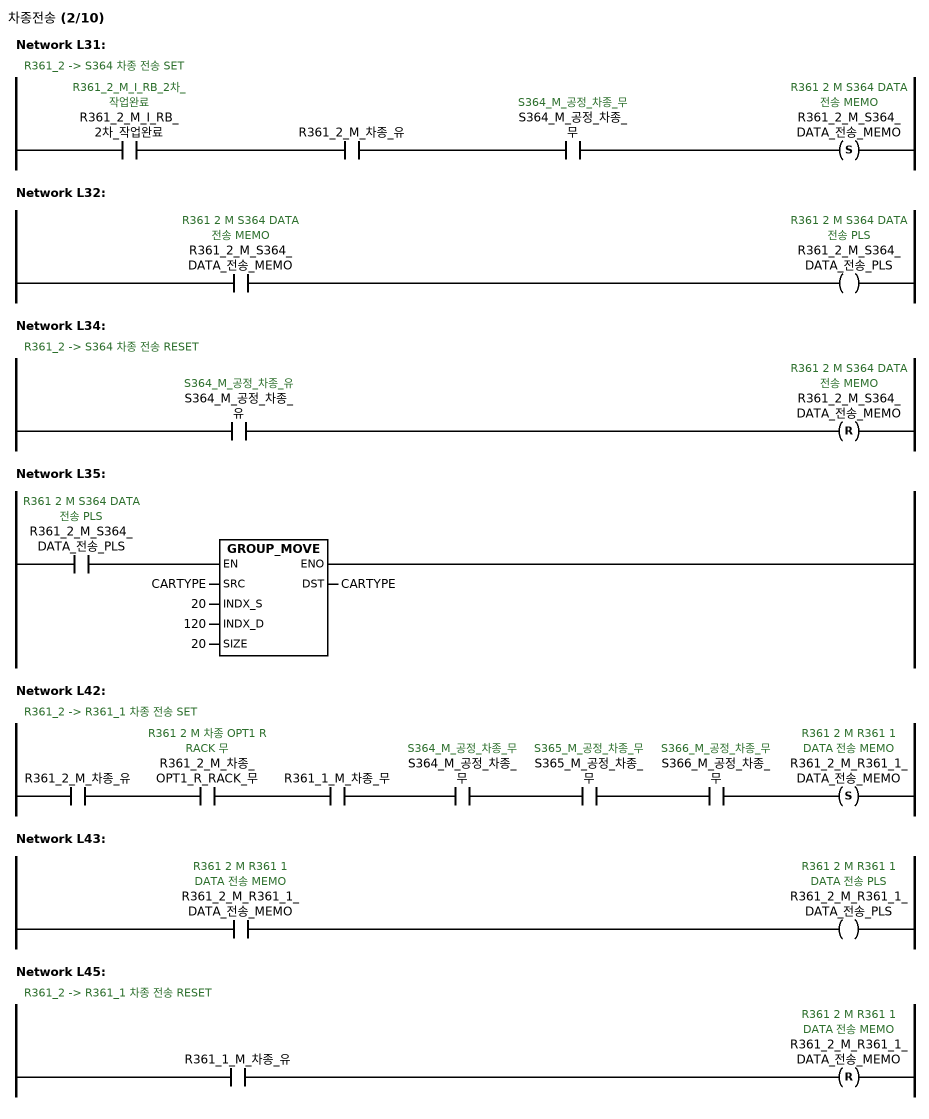
(* R361_2 -> S364 차종 전송 SET *)
(* Rung L31 *)
IF R361_2_M_I_RB_2차_작업완료 AND R361_2_M_차종_유 AND S364_M_공정_차종_무 THEN
    R361_2_M_S364_DATA_전송_MEMO := TRUE;
END_IF;
(* Rung L32 *)
R361_2_M_S364_DATA_전송_PLS := R361_2_M_S364_DATA_전송_MEMO;
(* R361_2 -> S364 차종 전송 RESET *)
(* Rung L34 *)
IF S364_M_공정_차종_유 THEN R361_2_M_S364_DATA_전송_MEMO := FALSE; END_IF;
(* Rung L35 *)
IF R361_2_M_S364_DATA_전송_PLS THEN
    CARTYPE := GROUP_MOVE(SRC := CARTYPE, INDX_S := 20, INDX_D := 120, SIZE := 20);
END_IF;
(* R361_2 -> R361_1 차종 전송 SET *)
(* Rung L42 *)
IF R361_2_M_차종_유 AND R361_2_M_차종_OPT1_R_RACK_무 AND R361_1_M_차종_무 AND S364_M_공정_차종_무 AND S365_M_공정_차종_무 AND S366_M_공정_차종_무 THEN
    R361_2_M_R361_1_DATA_전송_MEMO := TRUE;
END_IF;
(* Rung L43 *)
R361_2_M_R361_1_DATA_전송_PLS := R361_2_M_R361_1_DATA_전송_MEMO;
(* R361_2 -> R361_1 차종 전송 RESET *)
(* Rung L45 *)
IF R361_1_M_차종_유 THEN R361_2_M_R361_1_DATA_전송_MEMO := FALSE; END_IF;

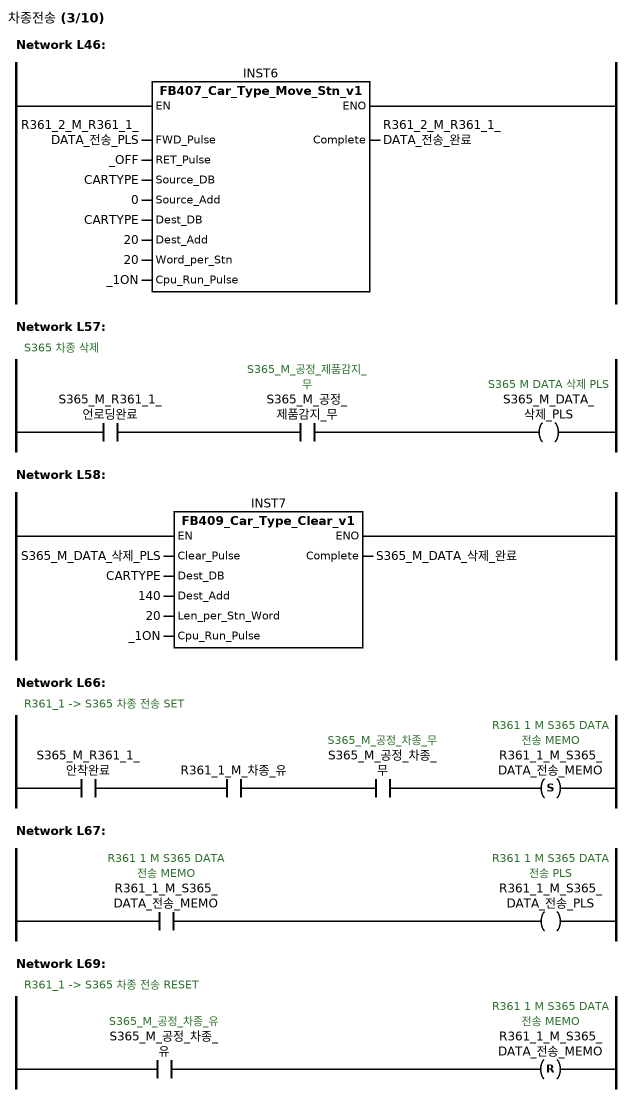
(* Rung L46 *)
INST6(FWD_Pulse := R361_2_M_R361_1_DATA_전송_PLS, RET_Pulse := _OFF, Source_DB := CARTYPE, Source_Add := 0, Dest_DB := CARTYPE, Dest_Add := 20, Word_per_Stn := 20, Cpu_Run_Pulse := _1ON, Complete => R361_2_M_R361_1_DATA_전송_완료);
(* S365 차종 삭제 *)
(* Rung L57 *)
S365_M_DATA_삭제_PLS := S365_M_R361_1_언로딩완료 AND S365_M_공정_제품감지_무;
(* Rung L58 *)
INST7(Clear_Pulse := S365_M_DATA_삭제_PLS, Dest_DB := CARTYPE, Dest_Add := 140, Len_per_Stn_Word := 20, Cpu_Run_Pulse := _1ON, Complete => S365_M_DATA_삭제_완료);
(* R361_1 -> S365 차종 전송 SET *)
(* Rung L66 *)
IF S365_M_R361_1_안착완료 AND R361_1_M_차종_유 AND S365_M_공정_차종_무 THEN
    R361_1_M_S365_DATA_전송_MEMO := TRUE;
END_IF;
(* Rung L67 *)
R361_1_M_S365_DATA_전송_PLS := R361_1_M_S365_DATA_전송_MEMO;
(* R361_1 -> S365 차종 전송 RESET *)
(* Rung L69 *)
IF S365_M_공정_차종_유 THEN R361_1_M_S365_DATA_전송_MEMO := FALSE; END_IF;

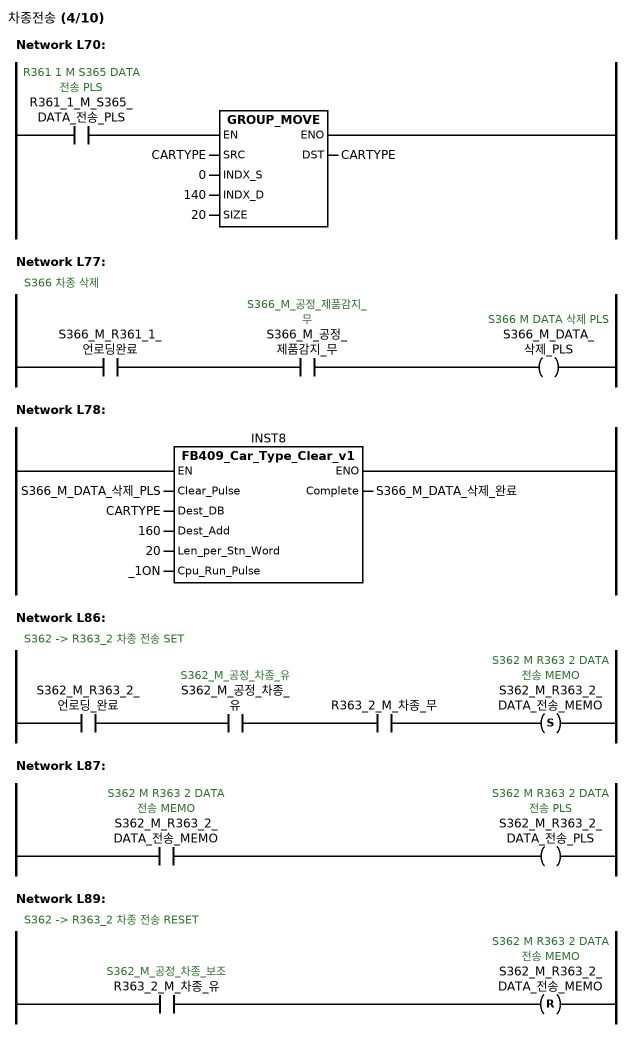
(* Rung L70 *)
IF R361_1_M_S365_DATA_전송_PLS THEN
    CARTYPE := GROUP_MOVE(SRC := CARTYPE, INDX_S := 0, INDX_D := 140, SIZE := 20);
END_IF;
(* S366 차종 삭제 *)
(* Rung L77 *)
S366_M_DATA_삭제_PLS := S366_M_R361_1_언로딩완료 AND S366_M_공정_제품감지_무;
(* Rung L78 *)
INST8(Clear_Pulse := S366_M_DATA_삭제_PLS, Dest_DB := CARTYPE, Dest_Add := 160, Len_per_Stn_Word := 20, Cpu_Run_Pulse := _1ON, Complete => S366_M_DATA_삭제_완료);
(* S362 -> R363_2 차종 전송 SET *)
(* Rung L86 *)
IF S362_M_R363_2_언로딩_완료 AND S362_M_공정_차종_유 AND R363_2_M_차종_무 THEN
    S362_M_R363_2_DATA_전송_MEMO := TRUE;
END_IF;
(* Rung L87 *)
S362_M_R363_2_DATA_전송_PLS := S362_M_R363_2_DATA_전송_MEMO;
(* S362 -> R363_2 차종 전송 RESET *)
(* Rung L89 *)
IF R363_2_M_차종_유 THEN S362_M_R363_2_DATA_전송_MEMO := FALSE; END_IF;

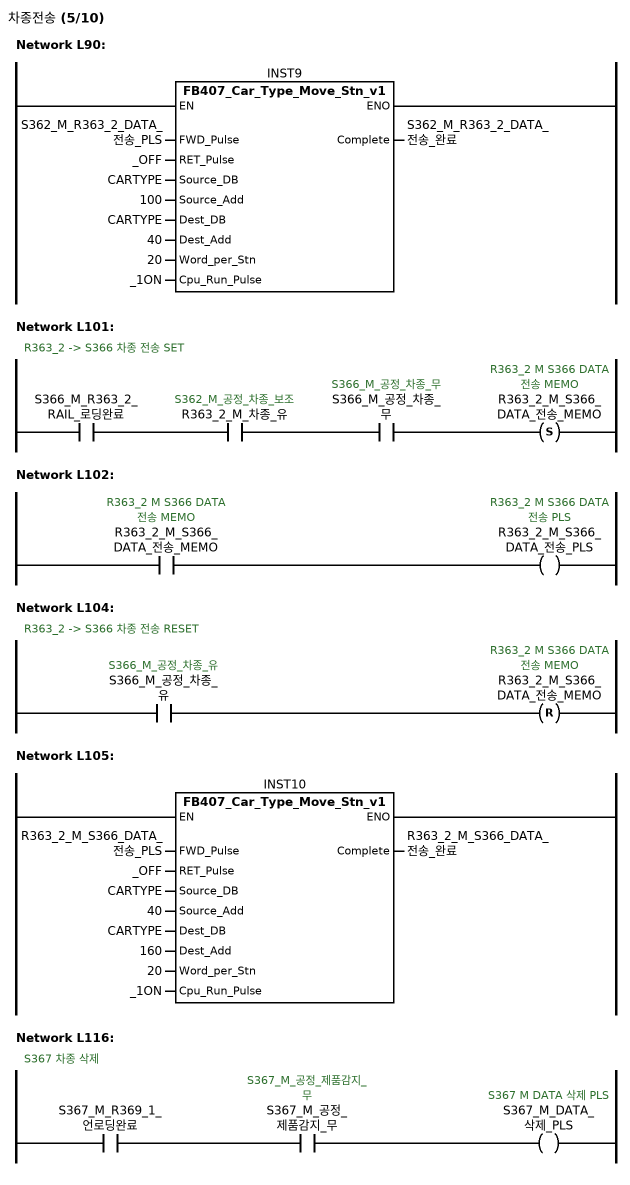
(* Rung L90 *)
INST9(FWD_Pulse := S362_M_R363_2_DATA_전송_PLS, RET_Pulse := _OFF, Source_DB := CARTYPE, Source_Add := 100, Dest_DB := CARTYPE, Dest_Add := 40, Word_per_Stn := 20, Cpu_Run_Pulse := _1ON, Complete => S362_M_R363_2_DATA_전송_완료);
(* R363_2 -> S366 차종 전송 SET *)
(* Rung L101 *)
IF S366_M_R363_2_RAIL_로딩완료 AND R363_2_M_차종_유 AND S366_M_공정_차종_무 THEN
    R363_2_M_S366_DATA_전송_MEMO := TRUE;
END_IF;
(* Rung L102 *)
R363_2_M_S366_DATA_전송_PLS := R363_2_M_S366_DATA_전송_MEMO;
(* R363_2 -> S366 차종 전송 RESET *)
(* Rung L104 *)
IF S366_M_공정_차종_유 THEN R363_2_M_S366_DATA_전송_MEMO := FALSE; END_IF;
(* Rung L105 *)
INST10(FWD_Pulse := R363_2_M_S366_DATA_전송_PLS, RET_Pulse := _OFF, Source_DB := CARTYPE, Source_Add := 40, Dest_DB := CARTYPE, Dest_Add := 160, Word_per_Stn := 20, Cpu_Run_Pulse := _1ON, Complete => R363_2_M_S366_DATA_전송_완료);
(* S367 차종 삭제 *)
(* Rung L116 *)
S367_M_DATA_삭제_PLS := S367_M_R369_1_언로딩완료 AND S367_M_공정_제품감지_무;

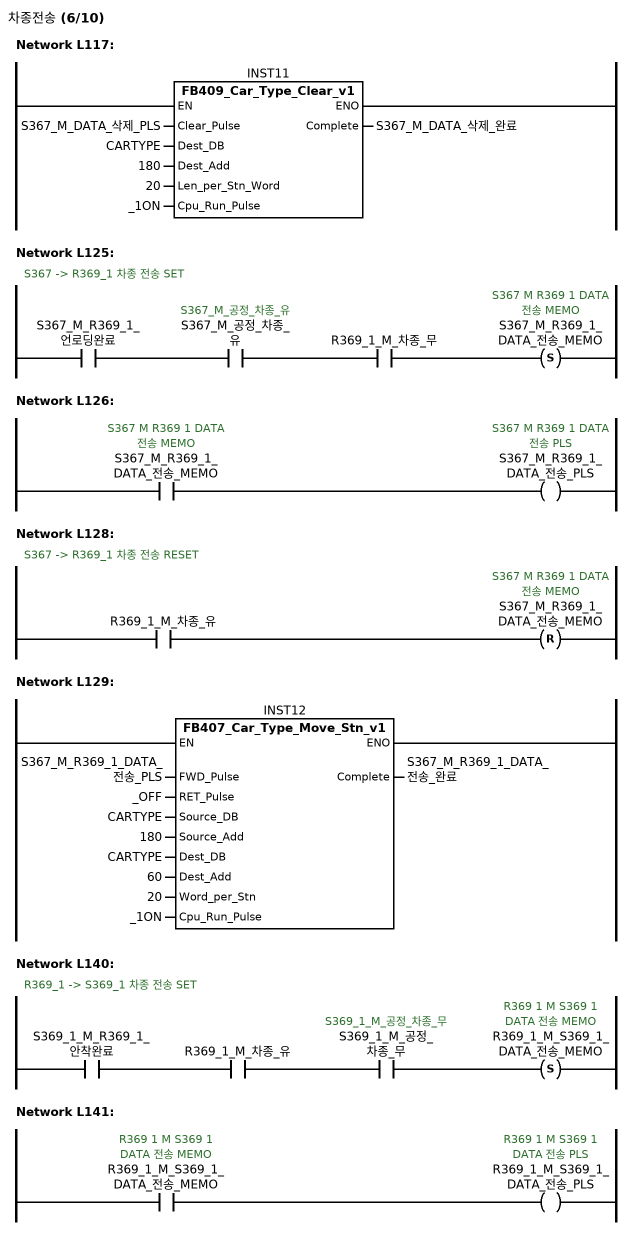
(* Rung L117 *)
INST11(Clear_Pulse := S367_M_DATA_삭제_PLS, Dest_DB := CARTYPE, Dest_Add := 180, Len_per_Stn_Word := 20, Cpu_Run_Pulse := _1ON, Complete => S367_M_DATA_삭제_완료);
(* S367 -> R369_1 차종 전송 SET *)
(* Rung L125 *)
IF S367_M_R369_1_언로딩완료 AND S367_M_공정_차종_유 AND R369_1_M_차종_무 THEN
    S367_M_R369_1_DATA_전송_MEMO := TRUE;
END_IF;
(* Rung L126 *)
S367_M_R369_1_DATA_전송_PLS := S367_M_R369_1_DATA_전송_MEMO;
(* S367 -> R369_1 차종 전송 RESET *)
(* Rung L128 *)
IF R369_1_M_차종_유 THEN S367_M_R369_1_DATA_전송_MEMO := FALSE; END_IF;
(* Rung L129 *)
INST12(FWD_Pulse := S367_M_R369_1_DATA_전송_PLS, RET_Pulse := _OFF, Source_DB := CARTYPE, Source_Add := 180, Dest_DB := CARTYPE, Dest_Add := 60, Word_per_Stn := 20, Cpu_Run_Pulse := _1ON, Complete => S367_M_R369_1_DATA_전송_완료);
(* R369_1 -> S369_1 차종 전송 SET *)
(* Rung L140 *)
IF S369_1_M_R369_1_안착완료 AND R369_1_M_차종_유 AND S369_1_M_공정_차종_무 THEN
    R369_1_M_S369_1_DATA_전송_MEMO := TRUE;
END_IF;
(* Rung L141 *)
R369_1_M_S369_1_DATA_전송_PLS := R369_1_M_S369_1_DATA_전송_MEMO;

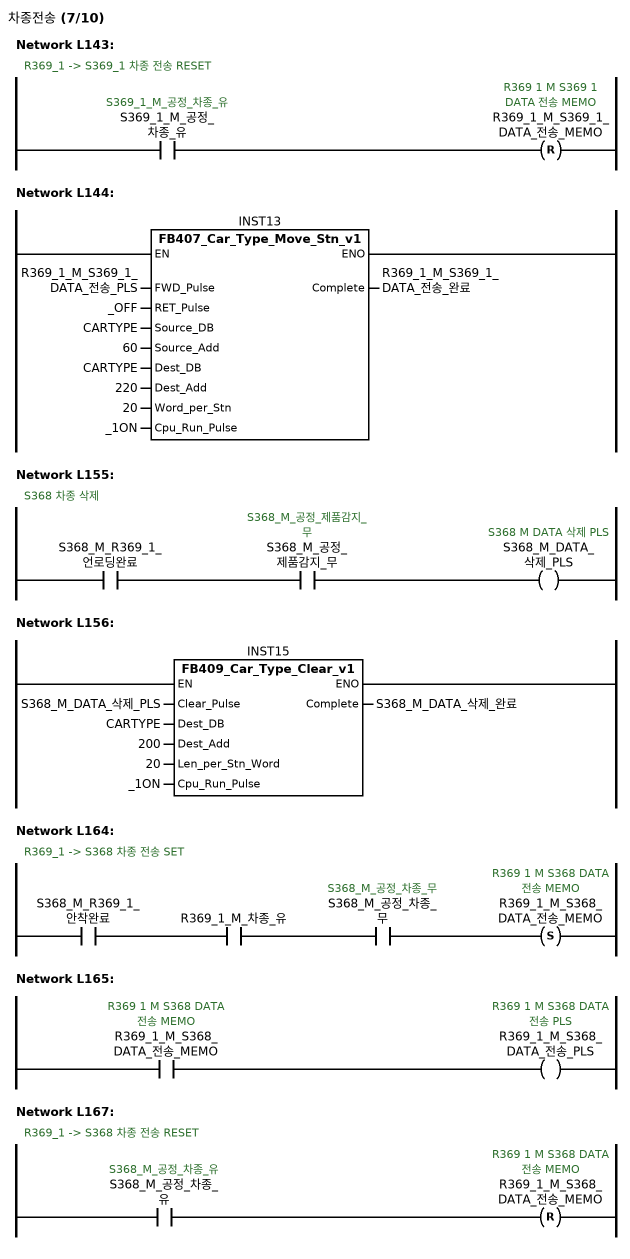
(* R369_1 -> S369_1 차종 전송 RESET *)
(* Rung L143 *)
IF S369_1_M_공정_차종_유 THEN R369_1_M_S369_1_DATA_전송_MEMO := FALSE; END_IF;
(* Rung L144 *)
INST13(FWD_Pulse := R369_1_M_S369_1_DATA_전송_PLS, RET_Pulse := _OFF, Source_DB := CARTYPE, Source_Add := 60, Dest_DB := CARTYPE, Dest_Add := 220, Word_per_Stn := 20, Cpu_Run_Pulse := _1ON, Complete => R369_1_M_S369_1_DATA_전송_완료);
(* S368 차종 삭제 *)
(* Rung L155 *)
S368_M_DATA_삭제_PLS := S368_M_R369_1_언로딩완료 AND S368_M_공정_제품감지_무;
(* Rung L156 *)
INST15(Clear_Pulse := S368_M_DATA_삭제_PLS, Dest_DB := CARTYPE, Dest_Add := 200, Len_per_Stn_Word := 20, Cpu_Run_Pulse := _1ON, Complete => S368_M_DATA_삭제_완료);
(* R369_1 -> S368 차종 전송 SET *)
(* Rung L164 *)
IF S368_M_R369_1_안착완료 AND R369_1_M_차종_유 AND S368_M_공정_차종_무 THEN
    R369_1_M_S368_DATA_전송_MEMO := TRUE;
END_IF;
(* Rung L165 *)
R369_1_M_S368_DATA_전송_PLS := R369_1_M_S368_DATA_전송_MEMO;
(* R369_1 -> S368 차종 전송 RESET *)
(* Rung L167 *)
IF S368_M_공정_차종_유 THEN R369_1_M_S368_DATA_전송_MEMO := FALSE; END_IF;

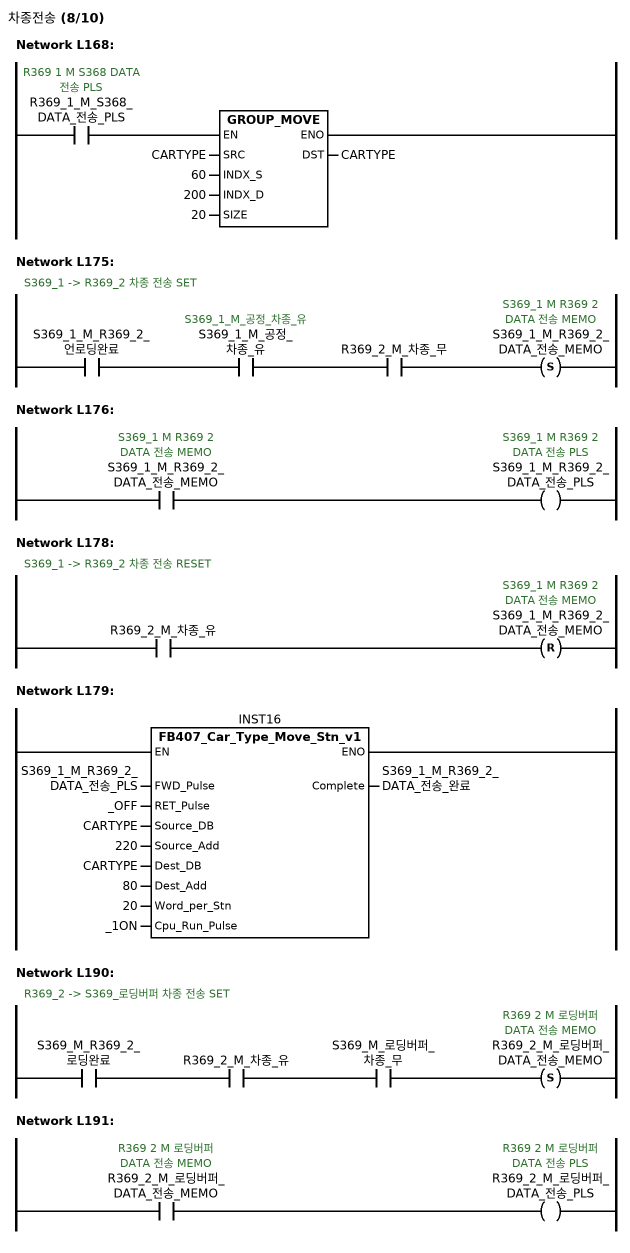
(* Rung L168 *)
IF R369_1_M_S368_DATA_전송_PLS THEN
    CARTYPE := GROUP_MOVE(SRC := CARTYPE, INDX_S := 60, INDX_D := 200, SIZE := 20);
END_IF;
(* S369_1 -> R369_2 차종 전송 SET *)
(* Rung L175 *)
IF S369_1_M_R369_2_언로딩완료 AND S369_1_M_공정_차종_유 AND R369_2_M_차종_무 THEN
    S369_1_M_R369_2_DATA_전송_MEMO := TRUE;
END_IF;
(* Rung L176 *)
S369_1_M_R369_2_DATA_전송_PLS := S369_1_M_R369_2_DATA_전송_MEMO;
(* S369_1 -> R369_2 차종 전송 RESET *)
(* Rung L178 *)
IF R369_2_M_차종_유 THEN S369_1_M_R369_2_DATA_전송_MEMO := FALSE; END_IF;
(* Rung L179 *)
INST16(FWD_Pulse := S369_1_M_R369_2_DATA_전송_PLS, RET_Pulse := _OFF, Source_DB := CARTYPE, Source_Add := 220, Dest_DB := CARTYPE, Dest_Add := 80, Word_per_Stn := 20, Cpu_Run_Pulse := _1ON, Complete => S369_1_M_R369_2_DATA_전송_완료);
(* R369_2 -> S369_로딩버퍼 차종 전송 SET *)
(* Rung L190 *)
IF S369_M_R369_2_로딩완료 AND R369_2_M_차종_유 AND S369_M_로딩버퍼_차종_무 THEN
    R369_2_M_로딩버퍼_DATA_전송_MEMO := TRUE;
END_IF;
(* Rung L191 *)
R369_2_M_로딩버퍼_DATA_전송_PLS := R369_2_M_로딩버퍼_DATA_전송_MEMO;

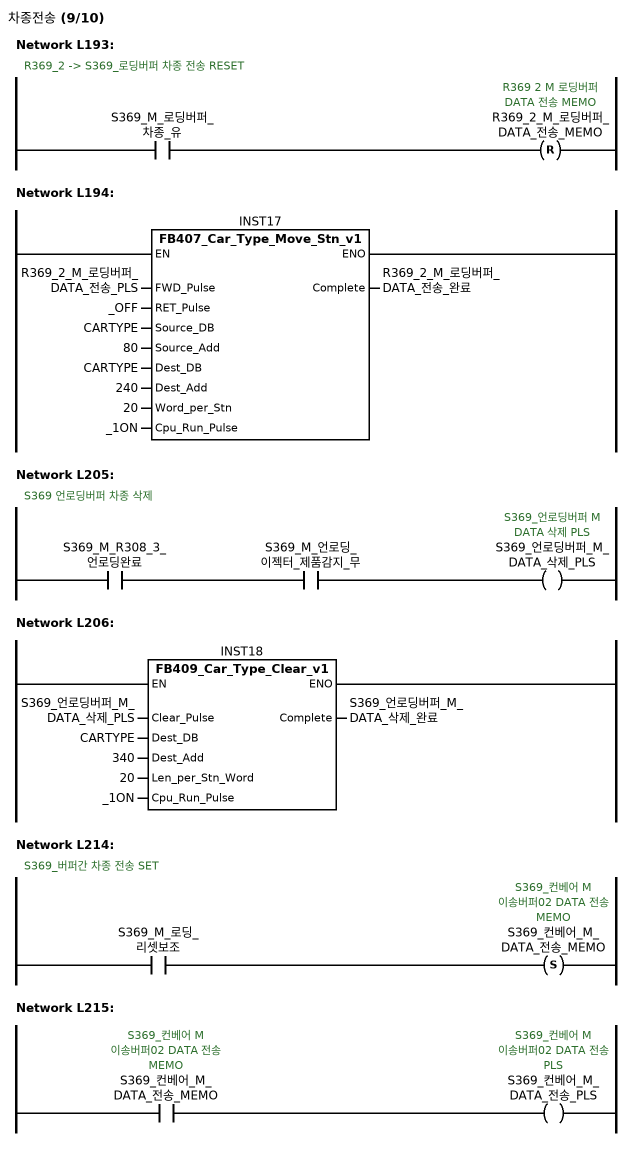
(* R369_2 -> S369_로딩버퍼 차종 전송 RESET *)
(* Rung L193 *)
IF S369_M_로딩버퍼_차종_유 THEN R369_2_M_로딩버퍼_DATA_전송_MEMO := FALSE; END_IF;
(* Rung L194 *)
INST17(FWD_Pulse := R369_2_M_로딩버퍼_DATA_전송_PLS, RET_Pulse := _OFF, Source_DB := CARTYPE, Source_Add := 80, Dest_DB := CARTYPE, Dest_Add := 240, Word_per_Stn := 20, Cpu_Run_Pulse := _1ON, Complete => R369_2_M_로딩버퍼_DATA_전송_완료);
(* S369 언로딩버퍼 차종 삭제 *)
(* Rung L205 *)
S369_언로딩버퍼_M_DATA_삭제_PLS := S369_M_R308_3_언로딩완료 AND S369_M_언로딩_이젝터_제품감지_무;
(* Rung L206 *)
INST18(Clear_Pulse := S369_언로딩버퍼_M_DATA_삭제_PLS, Dest_DB := CARTYPE, Dest_Add := 340, Len_per_Stn_Word := 20, Cpu_Run_Pulse := _1ON, Complete => S369_언로딩버퍼_M_DATA_삭제_완료);
(* S369_버퍼간 차종 전송 SET *)
(* Rung L214 *)
IF S369_M_로딩_리셋보조 THEN S369_컨베어_M_DATA_전송_MEMO := TRUE; END_IF;
(* Rung L215 *)
S369_컨베어_M_DATA_전송_PLS := S369_컨베어_M_DATA_전송_MEMO;

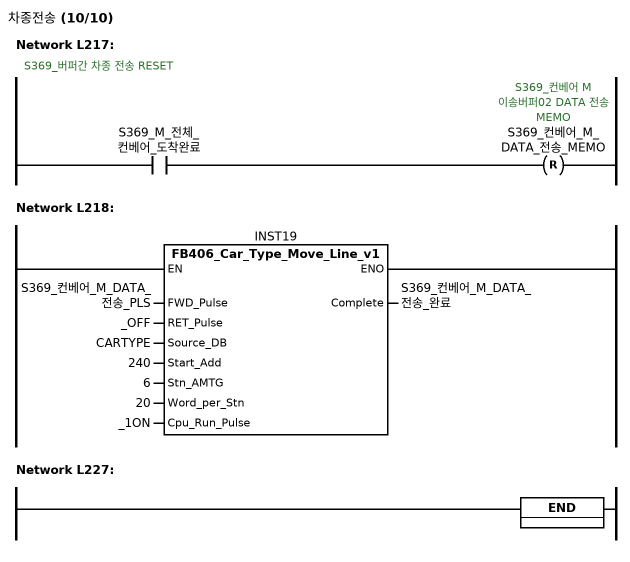
(* S369_버퍼간 차종 전송 RESET *)
(* Rung L217 *)
IF S369_M_전체_컨베어_도착완료 THEN S369_컨베어_M_DATA_전송_MEMO := FALSE; END_IF;
(* Rung L218 *)
INST19(FWD_Pulse := S369_컨베어_M_DATA_전송_PLS, RET_Pulse := _OFF, Source_DB := CARTYPE, Start_Add := 240, Stn_AMTG := 6, Word_per_Stn := 20, Cpu_Run_Pulse := _1ON, Complete => S369_컨베어_M_DATA_전송_완료);
(* Rung L227 *)
END();
END_PROGRAM

PROGRAM 알람트래킹 (* task: 스캔 프로그램 *)

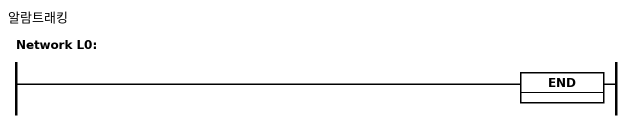
(* Rung L0 *)
END();
END_PROGRAM